RoboDK station: wcs_plc_20240624_150000.rdk

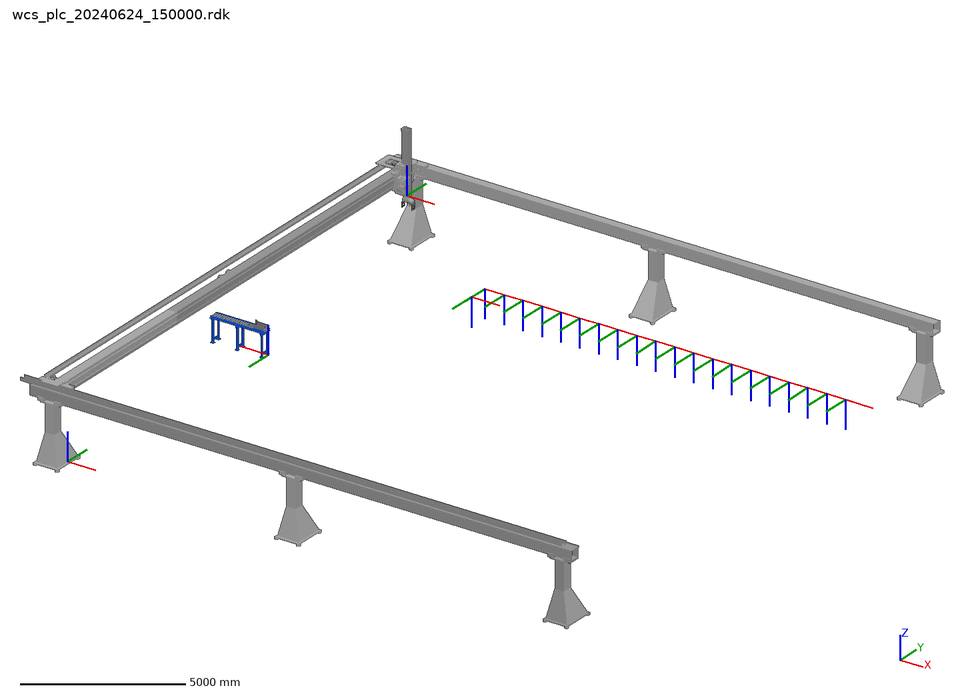
[picture v0: the station drawn from its stored meshes, robots at their saved joint values, targets as dots, program paths as lines]
Station wcs_plc_20240624_150000 (saved by RoboDK 5.6.8). Poses are relative to the parent item; angles as X-Y-Z fixed-axis rotations.
Station parameters (name, value as stored): TAGS, ['Milling']
  - frame conveyor Base at (750, 9500, 0) mm, rotated rx 0 ry 0 rz 180 deg
    - robot conveyor: 1 axes
        modified DH rows (alpha deg, a mm, theta deg, d mm): 0, 0, 0, 0 linear
        base shift (0, 0, 0) mm, rotated rx 0 ry 90 rz 0 deg
        joint limits [-99999] to [9999999]; home [0]; saved at [1000]
      - tool conveyor_TCP, TCP at (160, 110, 135) mm, rotated rx -180 ry 0 rz -180 deg
    - target con_pitch (joint target) at (1000, 0, 880) mm; joints [1000, 0, 0] of conveyor
    - target con_home (joint target) at (160, 110, 1015) mm, rotated rx -180 ry 0 rz -180 deg; joints [0] of conveyor
  - camera Camera 1
  - frame Frame 36 at (28300, 9440, 4940) mm, rotated rx -108 ry 0 rz 90 deg
  - frame gantry Base at (0, 0, 0) mm
    - robot gantry: 3 axes
        modified DH rows (alpha deg, a mm, theta deg, d mm): 0, 0, 0, 0 linear; 90, 0, 90, 0 linear; 90, 0, 0, 0 linear
        base shift (0, 0, 0) mm, rotated rx 0 ry -90 rz 180 deg
        joint limits [-5, -5, -5] to [18000, 17000, 1500]; home [0, 0, 0]; saved at [0, 0, 0]
      - frame gripper Base at (0, 0, 0) mm, rotated rx -180 ry 0 rz 0 deg
        - robot gripper: 1 axes
            modified DH rows (alpha deg, a mm, theta deg, d mm): 0, 0, 0, 0 linear
            base shift (0, 0, 0) mm, rotated rx 0 ry 90 rz 0 deg
            joint limits [-200] to [0]; home [0]; saved at [0]
        - target open_gripper (Cartesian target) at (0, 0, 0) mm; joints [0] of gripper
        - target close_gripper (Cartesian target) at (-55, 0, 0) mm; joints [-55] of gripper
      - tool gripper_TCP, TCP at (0, 0, 260) mm
    - target gantry_home (Cartesian target) at (-66.33, 17957.34, 1743.56) mm, rotated rx 180 ry 0 rz 0 deg; joints [0, 0, 0] of gantry
    - target UP_pickup (Cartesian target) at (590, 9400, 1743.56) mm, rotated rx 180 ry 0 rz 0 deg; joints [656.33, 8557.342, 0] of gantry
    - target IN_pickup (Cartesian target) at (590, 9400, 1275) mm, rotated rx 180 ry 0 rz 0 deg; joints [656.33, 8557.34, 468.56] of gantry
    - folder pallet
      - frame TeachingPoints_01-01-01 at (3833.67, 16507.34, 288.56) mm, rotated rx 180 ry 0 rz 0 deg
        - target Point_01-01-01 (Cartesian target) at (0, 0, 0) mm; joints [3900, 1450, 1195] of gantry
      - frame TeachingPoints_02-01-01 at (4533.67, 16507.34, 288.56) mm, rotated rx 180 ry 0 rz 0 deg
        - target Point_02-01-01 (Cartesian target) at (0, 0, 0) mm; joints [4600, 1450, 1195] of gantry
      - frame TeachingPoints_03-01-01 at (5233.67, 16507.34, 288.56) mm, rotated rx 180 ry 0 rz 0 deg
        - target Point_03-01-01 (Cartesian target) at (0, 0, 0) mm; joints [5300, 1450, 1195] of gantry
      - frame TeachingPoints_04-01-01 at (5933.67, 16507.34, 288.56) mm, rotated rx 180 ry 0 rz 0 deg
        - target Point_04-01-01 (Cartesian target) at (0, 0, 0) mm; joints [6000, 1450, 1195] of gantry
      - frame TeachingPoints_05-01-01 at (6633.67, 16507.34, 288.56) mm, rotated rx 180 ry 0 rz 0 deg
        - target Point_05-01-01 (Cartesian target) at (0, 0, 0) mm; joints [6700, 1450, 1195] of gantry
      - frame TeachingPoints_06-01-01 at (7333.67, 16507.34, 288.56) mm, rotated rx 180 ry 0 rz 0 deg
        - target Point_06-01-01 (Cartesian target) at (0, 0, 0) mm; joints [7400, 1450, 1195] of gantry
      - frame TeachingPoints_07-01-01 at (8033.67, 16507.34, 288.56) mm, rotated rx 180 ry 0 rz 0 deg
        - target Point_07-01-01 (Cartesian target) at (0, 0, 0) mm; joints [8100, 1450, 1195] of gantry
      - frame TeachingPoints_08-01-01 at (8733.67, 16507.34, 288.56) mm, rotated rx 180 ry 0 rz 0 deg
        - target Point_08-01-01 (Cartesian target) at (0, 0, 0) mm; joints [8800, 1450, 1195] of gantry
      - frame TeachingPoints_09-01-01 at (9433.67, 16507.34, 288.56) mm, rotated rx 180 ry 0 rz 0 deg
        - target Point_09-01-01 (Cartesian target) at (0, 0, 0) mm; joints [9500, 1450, 1195] of gantry
      - frame TeachingPoints_10-01-01 at (10133.67, 16507.34, 288.56) mm, rotated rx 180 ry 0 rz 0 deg
        - target Point_10-01-01 (Cartesian target) at (0, 0, 0) mm; joints [10200, 1450, 1195] of gantry
      - frame TeachingPoints_11-01-01 at (10833.67, 16507.34, 288.56) mm, rotated rx 180 ry 0 rz 0 deg
        - target Point_11-01-01 (Cartesian target) at (0, 0, 0) mm; joints [10900, 1450, 1195] of gantry
      - frame TeachingPoints_12-01-01 at (11533.67, 16507.34, 288.56) mm, rotated rx 180 ry 0 rz 0 deg
        - target Point_12-01-01 (Cartesian target) at (0, 0, 0) mm; joints [11600, 1450, 1195] of gantry
      - frame TeachingPoints_13-01-01 at (12233.67, 16507.34, 288.56) mm, rotated rx 180 ry 0 rz 0 deg
        - target Point_13-01-01 (Cartesian target) at (0, 0, 0) mm; joints [12300, 1450, 1195] of gantry
      - frame TeachingPoints_14-01-01 at (12933.67, 16507.34, 288.56) mm, rotated rx 180 ry 0 rz 0 deg
        - target Point_14-01-01 (Cartesian target) at (0, 0, 0) mm; joints [13000, 1450, 1195] of gantry
      - frame TeachingPoints_15-01-01 at (13633.67, 16507.34, 288.56) mm, rotated rx 180 ry 0 rz 0 deg
        - target Point_15-01-01 (Cartesian target) at (0, 0, 0) mm; joints [13700, 1450, 1195] of gantry
      - frame TeachingPoints_16-01-01 at (14333.67, 16507.34, 288.56) mm, rotated rx 180 ry 0 rz 0 deg
        - target Point_16-01-01 (Cartesian target) at (0, 0, 0) mm; joints [14400, 1450, 1195] of gantry
      - frame TeachingPoints_17-01-01 at (15033.67, 16507.34, 288.56) mm, rotated rx 180 ry 0 rz 0 deg
        - target Point_17-01-01 (Cartesian target) at (0, 0, 0) mm; joints [15100, 1450, 1195] of gantry
      - frame TeachingPoints_18-01-01 at (15733.67, 16507.34, 288.56) mm, rotated rx 180 ry 0 rz 0 deg
        - target Point_18-01-01 (Cartesian target) at (0, 0, 0) mm; joints [15800, 1450, 1195] of gantry
      - frame TeachingPoints_19-01-01 at (16433.67, 16507.34, 288.56) mm, rotated rx 180 ry 0 rz 0 deg
        - target Point_19-01-01 (Cartesian target) at (0, 0, 0) mm; joints [16500, 1450, 1195] of gantry
      - frame TeachingPoints_20-01-01 at (17133.67, 16507.34, 288.56) mm, rotated rx 180 ry 0 rz 0 deg
        - target Point_20-01-01 (Cartesian target) at (0, 0, 0) mm; joints [17200, 1450, 1195] of gantry
      - frame TeachingPoints_01-02-01 at (3833.67, 15807.34, 288.56) mm, rotated rx 180 ry 0 rz 0 deg
        - target Point_01-02-01 (Cartesian target) at (0, 0, 0) mm; joints [3900, 2150, 1195] of gantry
      - frame TeachingPoints_02-02-01 at (4533.67, 15807.34, 288.56) mm, rotated rx 180 ry 0 rz 0 deg
        - target Point_02-02-01 (Cartesian target) at (0, 0, 0) mm; joints [4600, 2150, 1195] of gantry
      - frame TeachingPoints_03-02-01 at (5233.67, 15807.34, 288.56) mm, rotated rx 180 ry 0 rz 0 deg
        - target Point_03-02-01 (Cartesian target) at (0, 0, 0) mm; joints [5300, 2150, 1195] of gantry
      - frame TeachingPoints_04-02-01 at (5933.67, 15807.34, 288.56) mm, rotated rx 180 ry 0 rz 0 deg
        - target Point_04-02-01 (Cartesian target) at (0, 0, 0) mm; joints [6000, 2150, 1195] of gantry
      - frame TeachingPoints_05-02-01 at (6633.67, 15807.34, 288.56) mm, rotated rx 180 ry 0 rz 0 deg
        - target Point_05-02-01 (Cartesian target) at (0, 0, 0) mm; joints [6700, 2150, 1195] of gantry
      - frame TeachingPoints_06-02-01 at (7333.67, 15807.34, 288.56) mm, rotated rx 180 ry 0 rz 0 deg
        - target Point_06-02-01 (Cartesian target) at (0, 0, 0) mm; joints [7400, 2150, 1195] of gantry
      - frame TeachingPoints_07-02-01 at (8033.67, 15807.34, 288.56) mm, rotated rx 180 ry 0 rz 0 deg
        - target Point_07-02-01 (Cartesian target) at (0, 0, 0) mm; joints [8100, 2150, 1195] of gantry
      - frame TeachingPoints_08-02-01 at (8733.67, 15807.34, 288.56) mm, rotated rx 180 ry 0 rz 0 deg
        - target Point_08-02-01 (Cartesian target) at (0, 0, 0) mm; joints [8800, 2150, 1195] of gantry
      - frame TeachingPoints_09-02-01 at (9433.67, 15807.34, 288.56) mm, rotated rx 180 ry 0 rz 0 deg
        - target Point_09-02-01 (Cartesian target) at (0, 0, 0) mm; joints [9500, 2150, 1195] of gantry
      - frame TeachingPoints_10-02-01 at (10133.67, 15807.34, 288.56) mm, rotated rx 180 ry 0 rz 0 deg
        - target Point_10-02-01 (Cartesian target) at (0, 0, 0) mm; joints [10200, 2150, 1195] of gantry
      - frame TeachingPoints_11-02-01 at (10833.67, 15807.34, 288.56) mm, rotated rx 180 ry 0 rz 0 deg
        - target Point_11-02-01 (Cartesian target) at (0, 0, 0) mm; joints [10900, 2150, 1195] of gantry
      - frame TeachingPoints_12-02-01 at (11533.67, 15807.34, 288.56) mm, rotated rx 180 ry 0 rz 0 deg
        - target Point_12-02-01 (Cartesian target) at (0, 0, 0) mm; joints [11600, 2150, 1195] of gantry
      - frame TeachingPoints_13-02-01 at (12233.67, 15807.34, 288.56) mm, rotated rx 180 ry 0 rz 0 deg
        - target Point_13-02-01 (Cartesian target) at (0, 0, 0) mm; joints [12300, 2150, 1195] of gantry
      - frame TeachingPoints_14-02-01 at (12933.67, 15807.34, 288.56) mm, rotated rx 180 ry 0 rz 0 deg
        - target Point_14-02-01 (Cartesian target) at (0, 0, 0) mm; joints [13000, 2150, 1195] of gantry
      - frame TeachingPoints_15-02-01 at (13633.67, 15807.34, 288.56) mm, rotated rx 180 ry 0 rz 0 deg
        - target Point_15-02-01 (Cartesian target) at (0, 0, 0) mm; joints [13700, 2150, 1195] of gantry
      - frame TeachingPoints_16-02-01 at (14333.67, 15807.34, 288.56) mm, rotated rx 180 ry 0 rz 0 deg
        - target Point_16-02-01 (Cartesian target) at (0, 0, 0) mm; joints [14400, 2150, 1195] of gantry
      - frame TeachingPoints_17-02-01 at (15033.67, 15807.34, 288.56) mm, rotated rx 180 ry 0 rz 0 deg
        - target Point_17-02-01 (Cartesian target) at (0, 0, 0) mm; joints [15100, 2150, 1195] of gantry
      - frame TeachingPoints_18-02-01 at (15733.67, 15807.34, 288.56) mm, rotated rx 180 ry 0 rz 0 deg
        - target Point_18-02-01 (Cartesian target) at (0, 0, 0) mm; joints [15800, 2150, 1195] of gantry
      - frame TeachingPoints_19-02-01 at (16433.67, 15807.34, 288.56) mm, rotated rx 180 ry 0 rz 0 deg
        - target Point_19-02-01 (Cartesian target) at (0, 0, 0) mm; joints [16500, 2150, 1195] of gantry
      - frame TeachingPoints_20-02-01 at (17133.67, 15807.34, 288.56) mm, rotated rx 180 ry 0 rz 0 deg
        - target Point_20-02-01 (Cartesian target) at (0, 0, 0) mm; joints [17200, 2150, 1195] of gantry
      - frame TeachingPoints_01-03-01 at (3833.67, 15107.34, 288.56) mm, rotated rx 180 ry 0 rz 0 deg
        - target Point_01-03-01 (Cartesian target) at (0, 0, 0) mm; joints [3900, 2850, 1195] of gantry
      - frame TeachingPoints_02-03-01 at (4533.67, 15107.34, 288.56) mm, rotated rx 180 ry 0 rz 0 deg
        - target Point_02-03-01 (Cartesian target) at (0, 0, 0) mm; joints [4600, 2850, 1195] of gantry
      - frame TeachingPoints_03-03-01 at (5233.67, 15107.34, 288.56) mm, rotated rx 180 ry 0 rz 0 deg
        - target Point_03-03-01 (Cartesian target) at (0, 0, 0) mm; joints [5300, 2850, 1195] of gantry
      - frame TeachingPoints_04-03-01 at (5933.67, 15107.34, 288.56) mm, rotated rx 180 ry 0 rz 0 deg
        - target Point_04-03-01 (Cartesian target) at (0, 0, 0) mm; joints [6000, 2850, 1195] of gantry
      - frame TeachingPoints_05-03-01 at (6633.67, 15107.34, 288.56) mm, rotated rx 180 ry 0 rz 0 deg
        - target Point_05-03-01 (Cartesian target) at (0, 0, 0) mm; joints [6700, 2850, 1195] of gantry
      - frame TeachingPoints_06-03-01 at (7333.67, 15107.34, 288.56) mm, rotated rx 180 ry 0 rz 0 deg
        - target Point_06-03-01 (Cartesian target) at (0, 0, 0) mm; joints [7400, 2850, 1195] of gantry
      - frame TeachingPoints_07-03-01 at (8033.67, 15107.34, 288.56) mm, rotated rx 180 ry 0 rz 0 deg
        - target Point_07-03-01 (Cartesian target) at (0, 0, 0) mm; joints [8100, 2850, 1195] of gantry
      - frame TeachingPoints_08-03-01 at (8733.67, 15107.34, 288.56) mm, rotated rx 180 ry 0 rz 0 deg
        - target Point_08-03-01 (Cartesian target) at (0, 0, 0) mm; joints [8800, 2850, 1195] of gantry
      - frame TeachingPoints_09-03-01 at (9433.67, 15107.34, 288.56) mm, rotated rx 180 ry 0 rz 0 deg
        - target Point_09-03-01 (Cartesian target) at (0, 0, 0) mm; joints [9500, 2850, 1195] of gantry
      - frame TeachingPoints_10-03-01 at (10133.67, 15107.34, 288.56) mm, rotated rx 180 ry 0 rz 0 deg
        - target Point_10-03-01 (Cartesian target) at (0, 0, 0) mm; joints [10200, 2850, 1195] of gantry
      - frame TeachingPoints_11-03-01 at (10833.67, 15107.34, 288.56) mm, rotated rx 180 ry 0 rz 0 deg
        - target Point_11-03-01 (Cartesian target) at (0, 0, 0) mm; joints [10900, 2850, 1195] of gantry
      - frame TeachingPoints_12-03-01 at (11533.67, 15107.34, 288.56) mm, rotated rx 180 ry 0 rz 0 deg
        - target Point_12-03-01 (Cartesian target) at (0, 0, 0) mm; joints [11600, 2850, 1195] of gantry
      - frame TeachingPoints_13-03-01 at (12233.67, 15107.34, 288.56) mm, rotated rx 180 ry 0 rz 0 deg
        - target Point_13-03-01 (Cartesian target) at (0, 0, 0) mm; joints [12300, 2850, 1195] of gantry
      - frame TeachingPoints_14-03-01 at (12933.67, 15107.34, 288.56) mm, rotated rx 180 ry 0 rz 0 deg
        - target Point_14-03-01 (Cartesian target) at (0, 0, 0) mm; joints [13000, 2850, 1195] of gantry
      - frame TeachingPoints_15-03-01 at (13633.67, 15107.34, 288.56) mm, rotated rx 180 ry 0 rz 0 deg
        - target Point_15-03-01 (Cartesian target) at (0, 0, 0) mm; joints [13700, 2850, 1195] of gantry
      - frame TeachingPoints_16-03-01 at (14333.67, 15107.34, 288.56) mm, rotated rx 180 ry 0 rz 0 deg
        - target Point_16-03-01 (Cartesian target) at (0, 0, 0) mm; joints [14400, 2850, 1195] of gantry
      - frame TeachingPoints_17-03-01 at (15033.67, 15107.34, 288.56) mm, rotated rx 180 ry 0 rz 0 deg
        - target Point_17-03-01 (Cartesian target) at (0, 0, 0) mm; joints [15100, 2850, 1195] of gantry
      - frame TeachingPoints_18-03-01 at (15733.67, 15107.34, 288.56) mm, rotated rx 180 ry 0 rz 0 deg
        - target Point_18-03-01 (Cartesian target) at (0, 0, 0) mm; joints [15800, 2850, 1195] of gantry
      - frame TeachingPoints_19-03-01 at (16433.67, 15107.34, 288.56) mm, rotated rx 180 ry 0 rz 0 deg
        - target Point_19-03-01 (Cartesian target) at (0, 0, 0) mm; joints [16500, 2850, 1195] of gantry
      - frame TeachingPoints_20-03-01 at (17133.67, 15107.34, 288.56) mm, rotated rx 180 ry 0 rz 0 deg
        - target Point_20-03-01 (Cartesian target) at (0, 0, 0) mm; joints [17200, 2850, 1195] of gantry
      - frame TeachingPoints_01-04-01 at (3833.67, 14407.34, 288.56) mm, rotated rx 180 ry 0 rz 0 deg
        - target Point_01-04-01 (Cartesian target) at (0, 0, 0) mm; joints [3900, 3550, 1195] of gantry
      - frame TeachingPoints_02-04-01 at (4533.67, 14407.34, 288.56) mm, rotated rx 180 ry 0 rz 0 deg
        - target Point_02-04-01 (Cartesian target) at (0, 0, 0) mm; joints [4600, 3550, 1195] of gantry
      - frame TeachingPoints_03-04-01 at (5233.67, 14407.34, 288.56) mm, rotated rx 180 ry 0 rz 0 deg
        - target Point_03-04-01 (Cartesian target) at (0, 0, 0) mm; joints [5300, 3550, 1195] of gantry
      - frame TeachingPoints_04-04-01 at (5933.67, 14407.34, 288.56) mm, rotated rx 180 ry 0 rz 0 deg
        - target Point_04-04-01 (Cartesian target) at (0, 0, 0) mm; joints [6000, 3550, 1195] of gantry
      - frame TeachingPoints_05-04-01 at (6633.67, 14407.34, 288.56) mm, rotated rx 180 ry 0 rz 0 deg
        - target Point_05-04-01 (Cartesian target) at (0, 0, 0) mm; joints [6700, 3550, 1195] of gantry
      - frame TeachingPoints_06-04-01 at (7333.67, 14407.34, 288.56) mm, rotated rx 180 ry 0 rz 0 deg
        - target Point_06-04-01 (Cartesian target) at (0, 0, 0) mm; joints [7400, 3550, 1195] of gantry
      - frame TeachingPoints_07-04-01 at (8033.67, 14407.34, 288.56) mm, rotated rx 180 ry 0 rz 0 deg
        - target Point_07-04-01 (Cartesian target) at (0, 0, 0) mm; joints [8100, 3550, 1195] of gantry
      - frame TeachingPoints_08-04-01 at (8733.67, 14407.34, 288.56) mm, rotated rx 180 ry 0 rz 0 deg
        - target Point_08-04-01 (Cartesian target) at (0, 0, 0) mm; joints [8800, 3550, 1195] of gantry
      - frame TeachingPoints_09-04-01 at (9433.67, 14407.34, 288.56) mm, rotated rx 180 ry 0 rz 0 deg
        - target Point_09-04-01 (Cartesian target) at (0, 0, 0) mm; joints [9500, 3550, 1195] of gantry
      - frame TeachingPoints_10-04-01 at (10133.67, 14407.34, 288.56) mm, rotated rx 180 ry 0 rz 0 deg
        - target Point_10-04-01 (Cartesian target) at (0, 0, 0) mm; joints [10200, 3550, 1195] of gantry
      - frame TeachingPoints_11-04-01 at (10833.67, 14407.34, 288.56) mm, rotated rx 180 ry 0 rz 0 deg
        - target Point_11-04-01 (Cartesian target) at (0, 0, 0) mm; joints [10900, 3550, 1195] of gantry
      - frame TeachingPoints_12-04-01 at (11533.67, 14407.34, 288.56) mm, rotated rx 180 ry 0 rz 0 deg
        - target Point_12-04-01 (Cartesian target) at (0, 0, 0) mm; joints [11600, 3550, 1195] of gantry
      - frame TeachingPoints_13-04-01 at (12233.67, 14407.34, 288.56) mm, rotated rx 180 ry 0 rz 0 deg
        - target Point_13-04-01 (Cartesian target) at (0, 0, 0) mm; joints [12300, 3550, 1195] of gantry
      - frame TeachingPoints_14-04-01 at (12933.67, 14407.34, 288.56) mm, rotated rx 180 ry 0 rz 0 deg
        - target Point_14-04-01 (Cartesian target) at (0, 0, 0) mm; joints [13000, 3550, 1195] of gantry
      - frame TeachingPoints_15-04-01 at (13633.67, 14407.34, 288.56) mm, rotated rx 180 ry 0 rz 0 deg
        - target Point_15-04-01 (Cartesian target) at (0, 0, 0) mm; joints [13700, 3550, 1195] of gantry
      - frame TeachingPoints_16-04-01 at (14333.67, 14407.34, 288.56) mm, rotated rx 180 ry 0 rz 0 deg
        - target Point_16-04-01 (Cartesian target) at (0, 0, 0) mm; joints [14400, 3550, 1195] of gantry
      - frame TeachingPoints_17-04-01 at (15033.67, 14407.34, 288.56) mm, rotated rx 180 ry 0 rz 0 deg
        - target Point_17-04-01 (Cartesian target) at (0, 0, 0) mm; joints [15100, 3550, 1195] of gantry
      - frame TeachingPoints_18-04-01 at (15733.67, 14407.34, 288.56) mm, rotated rx 180 ry 0 rz 0 deg
        - target Point_18-04-01 (Cartesian target) at (0, 0, 0) mm; joints [15800, 3550, 1195] of gantry
      - frame TeachingPoints_19-04-01 at (16433.67, 14407.34, 288.56) mm, rotated rx 180 ry 0 rz 0 deg
        - target Point_19-04-01 (Cartesian target) at (0, 0, 0) mm; joints [16500, 3550, 1195] of gantry
      - frame TeachingPoints_20-04-01 at (17133.67, 14407.34, 288.56) mm, rotated rx 180 ry 0 rz 0 deg
        - target Point_20-04-01 (Cartesian target) at (0, 0, 0) mm; joints [17200, 3550, 1195] of gantry
      - frame TeachingPoints_01-05-01 at (3833.67, 13707.34, 288.56) mm, rotated rx 180 ry 0 rz 0 deg
        - target Point_01-05-01 (Cartesian target) at (0, 0, 0) mm; joints [3900, 4250, 1195] of gantry
      - frame TeachingPoints_02-05-01 at (4533.67, 13707.34, 288.56) mm, rotated rx 180 ry 0 rz 0 deg
        - target Point_02-05-01 (Cartesian target) at (0, 0, 0) mm; joints [4600, 4250, 1195] of gantry
      - frame TeachingPoints_03-05-01 at (5233.67, 13707.34, 288.56) mm, rotated rx 180 ry 0 rz 0 deg
        - target Point_03-05-01 (Cartesian target) at (0, 0, 0) mm; joints [5300, 4250, 1195] of gantry
      - frame TeachingPoints_04-05-01 at (5933.67, 13707.34, 288.56) mm, rotated rx 180 ry 0 rz 0 deg
        - target Point_04-05-01 (Cartesian target) at (0, 0, 0) mm; joints [6000, 4250, 1195] of gantry
      - frame TeachingPoints_05-05-01 at (6633.67, 13707.34, 288.56) mm, rotated rx 180 ry 0 rz 0 deg
        - target Point_05-05-01 (Cartesian target) at (0, 0, 0) mm; joints [6700, 4250, 1195] of gantry
      - frame TeachingPoints_06-05-01 at (7333.67, 13707.34, 288.56) mm, rotated rx 180 ry 0 rz 0 deg
        - target Point_06-05-01 (Cartesian target) at (0, 0, 0) mm; joints [7400, 4250, 1195] of gantry
      - frame TeachingPoints_07-05-01 at (8033.67, 13707.34, 288.56) mm, rotated rx 180 ry 0 rz 0 deg
        - target Point_07-05-01 (Cartesian target) at (0, 0, 0) mm; joints [8100, 4250, 1195] of gantry
      - frame TeachingPoints_08-05-01 at (8733.67, 13707.34, 288.56) mm, rotated rx 180 ry 0 rz 0 deg
        - target Point_08-05-01 (Cartesian target) at (0, 0, 0) mm; joints [8800, 4250, 1195] of gantry
      - frame TeachingPoints_09-05-01 at (9433.67, 13707.34, 288.56) mm, rotated rx 180 ry 0 rz 0 deg
        - target Point_09-05-01 (Cartesian target) at (0, 0, 0) mm; joints [9500, 4250, 1195] of gantry
      - frame TeachingPoints_10-05-01 at (10133.67, 13707.34, 288.56) mm, rotated rx 180 ry 0 rz 0 deg
        - target Point_10-05-01 (Cartesian target) at (0, 0, 0) mm; joints [10200, 4250, 1195] of gantry
      - frame TeachingPoints_11-05-01 at (10833.67, 13707.34, 288.56) mm, rotated rx 180 ry 0 rz 0 deg
        - target Point_11-05-01 (Cartesian target) at (0, 0, 0) mm; joints [10900, 4250, 1195] of gantry
      - frame TeachingPoints_12-05-01 at (11533.67, 13707.34, 288.56) mm, rotated rx 180 ry 0 rz 0 deg
        - target Point_12-05-01 (Cartesian target) at (0, 0, 0) mm; joints [11600, 4250, 1195] of gantry
      - frame TeachingPoints_13-05-01 at (12233.67, 13707.34, 288.56) mm, rotated rx 180 ry 0 rz 0 deg
        - target Point_13-05-01 (Cartesian target) at (0, 0, 0) mm; joints [12300, 4250, 1195] of gantry
      - frame TeachingPoints_14-05-01 at (12933.67, 13707.34, 288.56) mm, rotated rx 180 ry 0 rz 0 deg
        - target Point_14-05-01 (Cartesian target) at (0, 0, 0) mm; joints [13000, 4250, 1195] of gantry
      - frame TeachingPoints_15-05-01 at (13633.67, 13707.34, 288.56) mm, rotated rx 180 ry 0 rz 0 deg
        - target Point_15-05-01 (Cartesian target) at (0, 0, 0) mm; joints [13700, 4250, 1195] of gantry
      - frame TeachingPoints_16-05-01 at (14333.67, 13707.34, 288.56) mm, rotated rx 180 ry 0 rz 0 deg
        - target Point_16-05-01 (Cartesian target) at (0, 0, 0) mm; joints [14400, 4250, 1195] of gantry
      - frame TeachingPoints_17-05-01 at (15033.67, 13707.34, 288.56) mm, rotated rx 180 ry 0 rz 0 deg
        - target Point_17-05-01 (Cartesian target) at (0, 0, 0) mm; joints [15100, 4250, 1195] of gantry
      - frame TeachingPoints_18-05-01 at (15733.67, 13707.34, 288.56) mm, rotated rx 180 ry 0 rz 0 deg
        - target Point_18-05-01 (Cartesian target) at (0, 0, 0) mm; joints [15800, 4250, 1195] of gantry
      - frame TeachingPoints_19-05-01 at (16433.67, 13707.34, 288.56) mm, rotated rx 180 ry 0 rz 0 deg
        - target Point_19-05-01 (Cartesian target) at (0, 0, 0) mm; joints [16500, 4250, 1195] of gantry
      - frame TeachingPoints_20-05-01 at (17133.67, 13707.34, 288.56) mm, rotated rx 180 ry 0 rz 0 deg
        - target Point_20-05-01 (Cartesian target) at (0, 0, 0) mm; joints [17200, 4250, 1195] of gantry
      - frame TeachingPoints_01-06-01 at (3833.67, 13007.34, 288.56) mm, rotated rx 180 ry 0 rz 0 deg
        - target Point_01-06-01 (Cartesian target) at (0, 0, 0) mm; joints [3900, 4950, 1195] of gantry
      - frame TeachingPoints_02-06-01 at (4533.67, 13007.34, 288.56) mm, rotated rx 180 ry 0 rz 0 deg
        - target Point_02-06-01 (Cartesian target) at (0, 0, 0) mm; joints [4600, 4950, 1195] of gantry
      - frame TeachingPoints_03-06-01 at (5233.67, 13007.34, 288.56) mm, rotated rx 180 ry 0 rz 0 deg
        - target Point_03-06-01 (Cartesian target) at (0, 0, 0) mm; joints [5300, 4950, 1195] of gantry
      - frame TeachingPoints_04-06-01 at (5933.67, 13007.34, 288.56) mm, rotated rx 180 ry 0 rz 0 deg
        - target Point_04-06-01 (Cartesian target) at (0, 0, 0) mm; joints [6000, 4950, 1195] of gantry
      - frame TeachingPoints_05-06-01 at (6633.67, 13007.34, 288.56) mm, rotated rx 180 ry 0 rz 0 deg
        - target Point_05-06-01 (Cartesian target) at (0, 0, 0) mm; joints [6700, 4950, 1195] of gantry
      - frame TeachingPoints_06-06-01 at (7333.67, 13007.34, 288.56) mm, rotated rx 180 ry 0 rz 0 deg
        - target Point_06-06-01 (Cartesian target) at (0, 0, 0) mm; joints [7400, 4950, 1195] of gantry
      - frame TeachingPoints_07-06-01 at (8033.67, 13007.34, 288.56) mm, rotated rx 180 ry 0 rz 0 deg
        - target Point_07-06-01 (Cartesian target) at (0, 0, 0) mm; joints [8100, 4950, 1195] of gantry
      - frame TeachingPoints_08-06-01 at (8733.67, 13007.34, 288.56) mm, rotated rx 180 ry 0 rz 0 deg
        - target Point_08-06-01 (Cartesian target) at (0, 0, 0) mm; joints [8800, 4950, 1195] of gantry
      - frame TeachingPoints_09-06-01 at (9433.67, 13007.34, 288.56) mm, rotated rx 180 ry 0 rz 0 deg
        - target Point_09-06-01 (Cartesian target) at (0, 0, 0) mm; joints [9500, 4950, 1195] of gantry
      - frame TeachingPoints_10-06-01 at (10133.67, 13007.34, 288.56) mm, rotated rx 180 ry 0 rz 0 deg
        - target Point_10-06-01 (Cartesian target) at (0, 0, 0) mm; joints [10200, 4950, 1195] of gantry
      - frame TeachingPoints_11-06-01 at (10833.67, 13007.34, 288.56) mm, rotated rx 180 ry 0 rz 0 deg
        - target Point_11-06-01 (Cartesian target) at (0, 0, 0) mm; joints [10900, 4950, 1195] of gantry
      - frame TeachingPoints_12-06-01 at (11533.67, 13007.34, 288.56) mm, rotated rx 180 ry 0 rz 0 deg
        - target Point_12-06-01 (Cartesian target) at (0, 0, 0) mm; joints [11600, 4950, 1195] of gantry
      - frame TeachingPoints_13-06-01 at (12233.67, 13007.34, 288.56) mm, rotated rx 180 ry 0 rz 0 deg
        - target Point_13-06-01 (Cartesian target) at (0, 0, 0) mm; joints [12300, 4950, 1195] of gantry
      - frame TeachingPoints_14-06-01 at (12933.67, 13007.34, 288.56) mm, rotated rx 180 ry 0 rz 0 deg
        - target Point_14-06-01 (Cartesian target) at (0, 0, 0) mm; joints [13000, 4950, 1195] of gantry
      - frame TeachingPoints_15-06-01 at (13633.67, 13007.34, 288.56) mm, rotated rx 180 ry 0 rz 0 deg
        - target Point_15-06-01 (Cartesian target) at (0, 0, 0) mm; joints [13700, 4950, 1195] of gantry
      - frame TeachingPoints_16-06-01 at (14333.67, 13007.34, 288.56) mm, rotated rx 180 ry 0 rz 0 deg
        - target Point_16-06-01 (Cartesian target) at (0, 0, 0) mm; joints [14400, 4950, 1195] of gantry
      - frame TeachingPoints_17-06-01 at (15033.67, 13007.34, 288.56) mm, rotated rx 180 ry 0 rz 0 deg
        - target Point_17-06-01 (Cartesian target) at (0, 0, 0) mm; joints [15100, 4950, 1195] of gantry
      - frame TeachingPoints_18-06-01 at (15733.67, 13007.34, 288.56) mm, rotated rx 180 ry 0 rz 0 deg
        - target Point_18-06-01 (Cartesian target) at (0, 0, 0) mm; joints [15800, 4950, 1195] of gantry
      - frame TeachingPoints_19-06-01 at (16433.67, 13007.34, 288.56) mm, rotated rx 180 ry 0 rz 0 deg
        - target Point_19-06-01 (Cartesian target) at (0, 0, 0) mm; joints [16500, 4950, 1195] of gantry
      - frame TeachingPoints_20-06-01 at (17133.67, 13007.34, 288.56) mm, rotated rx 180 ry 0 rz 0 deg
        - target Point_20-06-01 (Cartesian target) at (0, 0, 0) mm; joints [17200, 4950, 1195] of gantry
      - frame TeachingPoints_01-07-01 at (3833.67, 12307.34, 288.56) mm, rotated rx 180 ry 0 rz 0 deg
        - target Point_01-07-01 (Cartesian target) at (0, 0, 0) mm; joints [3900, 5650, 1195] of gantry
      - frame TeachingPoints_02-07-01 at (4533.67, 12307.34, 288.56) mm, rotated rx 180 ry 0 rz 0 deg
        - target Point_02-07-01 (Cartesian target) at (0, 0, 0) mm; joints [4600, 5650, 1195] of gantry
      - frame TeachingPoints_03-07-01 at (5233.67, 12307.34, 288.56) mm, rotated rx 180 ry 0 rz 0 deg
        - target Point_03-07-01 (Cartesian target) at (0, 0, 0) mm; joints [5300, 5650, 1195] of gantry
      - frame TeachingPoints_04-07-01 at (5933.67, 12307.34, 288.56) mm, rotated rx 180 ry 0 rz 0 deg
        - target Point_04-07-01 (Cartesian target) at (0, 0, 0) mm; joints [6000, 5650, 1195] of gantry
      - frame TeachingPoints_05-07-01 at (6633.67, 12307.34, 288.56) mm, rotated rx 180 ry 0 rz 0 deg
        - target Point_05-07-01 (Cartesian target) at (0, 0, 0) mm; joints [6700, 5650, 1195] of gantry
      - frame TeachingPoints_06-07-01 at (7333.67, 12307.34, 288.56) mm, rotated rx 180 ry 0 rz 0 deg
        - target Point_06-07-01 (Cartesian target) at (0, 0, 0) mm; joints [7400, 5650, 1195] of gantry
      - frame TeachingPoints_07-07-01 at (8033.67, 12307.34, 288.56) mm, rotated rx 180 ry 0 rz 0 deg
        - target Point_07-07-01 (Cartesian target) at (0, 0, 0) mm; joints [8100, 5650, 1195] of gantry
      - frame TeachingPoints_08-07-01 at (8733.67, 12307.34, 288.56) mm, rotated rx 180 ry 0 rz 0 deg
        - target Point_08-07-01 (Cartesian target) at (0, 0, 0) mm; joints [8800, 5650, 1195] of gantry
      - frame TeachingPoints_09-07-01 at (9433.67, 12307.34, 288.56) mm, rotated rx 180 ry 0 rz 0 deg
        - target Point_09-07-01 (Cartesian target) at (0, 0, 0) mm; joints [9500, 5650, 1195] of gantry
      - frame TeachingPoints_10-07-01 at (10133.67, 12307.34, 288.56) mm, rotated rx 180 ry 0 rz 0 deg
        - target Point_10-07-01 (Cartesian target) at (0, 0, 0) mm; joints [10200, 5650, 1195] of gantry
      - frame TeachingPoints_11-07-01 at (10833.67, 12307.34, 288.56) mm, rotated rx 180 ry 0 rz 0 deg
        - target Point_11-07-01 (Cartesian target) at (0, 0, 0) mm; joints [10900, 5650, 1195] of gantry
      - frame TeachingPoints_12-07-01 at (11533.67, 12307.34, 288.56) mm, rotated rx 180 ry 0 rz 0 deg
        - target Point_12-07-01 (Cartesian target) at (0, 0, 0) mm; joints [11600, 5650, 1195] of gantry
      - frame TeachingPoints_13-07-01 at (12233.67, 12307.34, 288.56) mm, rotated rx 180 ry 0 rz 0 deg
        - target Point_13-07-01 (Cartesian target) at (0, 0, 0) mm; joints [12300, 5650, 1195] of gantry
      - frame TeachingPoints_14-07-01 at (12933.67, 12307.34, 288.56) mm, rotated rx 180 ry 0 rz 0 deg
        - target Point_14-07-01 (Cartesian target) at (0, 0, 0) mm; joints [13000, 5650, 1195] of gantry
      - frame TeachingPoints_15-07-01 at (13633.67, 12307.34, 288.56) mm, rotated rx 180 ry 0 rz 0 deg
        - target Point_15-07-01 (Cartesian target) at (0, 0, 0) mm; joints [13700, 5650, 1195] of gantry
      - frame TeachingPoints_16-07-01 at (14333.67, 12307.34, 288.56) mm, rotated rx 180 ry 0 rz 0 deg
        - target Point_16-07-01 (Cartesian target) at (0, 0, 0) mm; joints [14400, 5650, 1195] of gantry
      - frame TeachingPoints_17-07-01 at (15033.67, 12307.34, 288.56) mm, rotated rx 180 ry 0 rz 0 deg
        - target Point_17-07-01 (Cartesian target) at (0, 0, 0) mm; joints [15100, 5650, 1195] of gantry
      - frame TeachingPoints_18-07-01 at (15733.67, 12307.34, 288.56) mm, rotated rx 180 ry 0 rz 0 deg
        - target Point_18-07-01 (Cartesian target) at (0, 0, 0) mm; joints [15800, 5650, 1195] of gantry
      - frame TeachingPoints_19-07-01 at (16433.67, 12307.34, 288.56) mm, rotated rx 180 ry 0 rz 0 deg
        - target Point_19-07-01 (Cartesian target) at (0, 0, 0) mm; joints [16500, 5650, 1195] of gantry
      - frame TeachingPoints_20-07-01 at (17133.67, 12307.34, 288.56) mm, rotated rx 180 ry 0 rz 0 deg
        - target Point_20-07-01 (Cartesian target) at (0, 0, 0) mm; joints [17200, 5650, 1195] of gantry
      - frame TeachingPoints_01-08-01 at (3833.67, 11607.34, 288.56) mm, rotated rx 180 ry 0 rz 0 deg
        - target Point_01-08-01 (Cartesian target) at (0, 0, 0) mm; joints [3900, 6350, 1195] of gantry
      - frame TeachingPoints_02-08-01 at (4533.67, 11607.34, 288.56) mm, rotated rx 180 ry 0 rz 0 deg
        - target Point_02-08-01 (Cartesian target) at (0, 0, 0) mm; joints [4600, 6350, 1195] of gantry
      - frame TeachingPoints_03-08-01 at (5233.67, 11607.34, 288.56) mm, rotated rx 180 ry 0 rz 0 deg
        - target Point_03-08-01 (Cartesian target) at (0, 0, 0) mm; joints [5300, 6350, 1195] of gantry
      - frame TeachingPoints_04-08-01 at (5933.67, 11607.34, 288.56) mm, rotated rx 180 ry 0 rz 0 deg
        - target Point_04-08-01 (Cartesian target) at (0, 0, 0) mm; joints [6000, 6350, 1195] of gantry
      - frame TeachingPoints_05-08-01 at (6633.67, 11607.34, 288.56) mm, rotated rx 180 ry 0 rz 0 deg
        - target Point_05-08-01 (Cartesian target) at (0, 0, 0) mm; joints [6700, 6350, 1195] of gantry
      - frame TeachingPoints_06-08-01 at (7333.67, 11607.34, 288.56) mm, rotated rx 180 ry 0 rz 0 deg
        - target Point_06-08-01 (Cartesian target) at (0, 0, 0) mm; joints [7400, 6350, 1195] of gantry
      - frame TeachingPoints_07-08-01 at (8033.67, 11607.34, 288.56) mm, rotated rx 180 ry 0 rz 0 deg
        - target Point_07-08-01 (Cartesian target) at (0, 0, 0) mm; joints [8100, 6350, 1195] of gantry
      - frame TeachingPoints_08-08-01 at (8733.67, 11607.34, 288.56) mm, rotated rx 180 ry 0 rz 0 deg
        - target Point_08-08-01 (Cartesian target) at (0, 0, 0) mm; joints [8800, 6350, 1195] of gantry
      - frame TeachingPoints_09-08-01 at (9433.67, 11607.34, 288.56) mm, rotated rx 180 ry 0 rz 0 deg
        - target Point_09-08-01 (Cartesian target) at (0, 0, 0) mm; joints [9500, 6350, 1195] of gantry
      - frame TeachingPoints_10-08-01 at (10133.67, 11607.34, 288.56) mm, rotated rx 180 ry 0 rz 0 deg
        - target Point_10-08-01 (Cartesian target) at (0, 0, 0) mm; joints [10200, 6350, 1195] of gantry
      - frame TeachingPoints_11-08-01 at (10833.67, 11607.34, 288.56) mm, rotated rx 180 ry 0 rz 0 deg
        - target Point_11-08-01 (Cartesian target) at (0, 0, 0) mm; joints [10900, 6350, 1195] of gantry
      - frame TeachingPoints_12-08-01 at (11533.67, 11607.34, 288.56) mm, rotated rx 180 ry 0 rz 0 deg
        - target Point_12-08-01 (Cartesian target) at (0, 0, 0) mm; joints [11600, 6350, 1195] of gantry
      - frame TeachingPoints_13-08-01 at (12233.67, 11607.34, 288.56) mm, rotated rx 180 ry 0 rz 0 deg
        - target Point_13-08-01 (Cartesian target) at (0, 0, 0) mm; joints [12300, 6350, 1195] of gantry
      - frame TeachingPoints_14-08-01 at (12933.67, 11607.34, 288.56) mm, rotated rx 180 ry 0 rz 0 deg
        - target Point_14-08-01 (Cartesian target) at (0, 0, 0) mm; joints [13000, 6350, 1195] of gantry
      - frame TeachingPoints_15-08-01 at (13633.67, 11607.34, 288.56) mm, rotated rx 180 ry 0 rz 0 deg
        - target Point_15-08-01 (Cartesian target) at (0, 0, 0) mm; joints [13700, 6350, 1195] of gantry
      - frame TeachingPoints_16-08-01 at (14333.67, 11607.34, 288.56) mm, rotated rx 180 ry 0 rz 0 deg
        - target Point_16-08-01 (Cartesian target) at (0, 0, 0) mm; joints [14400, 6350, 1195] of gantry
      - frame TeachingPoints_17-08-01 at (15033.67, 11607.34, 288.56) mm, rotated rx 180 ry 0 rz 0 deg
        - target Point_17-08-01 (Cartesian target) at (0, 0, 0) mm; joints [15100, 6350, 1195] of gantry
      - frame TeachingPoints_18-08-01 at (15733.67, 11607.34, 288.56) mm, rotated rx 180 ry 0 rz 0 deg
        - target Point_18-08-01 (Cartesian target) at (0, 0, 0) mm; joints [15800, 6350, 1195] of gantry
      - frame TeachingPoints_19-08-01 at (16433.67, 11607.34, 288.56) mm, rotated rx 180 ry 0 rz 0 deg
        - target Point_19-08-01 (Cartesian target) at (0, 0, 0) mm; joints [16500, 6350, 1195] of gantry
      - frame TeachingPoints_20-08-01 at (17133.67, 11607.34, 288.56) mm, rotated rx 180 ry 0 rz 0 deg
        - target Point_20-08-01 (Cartesian target) at (0, 0, 0) mm; joints [17200, 6350, 1195] of gantry
      - frame TeachingPoints_01-09-01 at (3833.67, 10907.34, 288.56) mm, rotated rx 180 ry 0 rz 0 deg
        - target Point_01-09-01 (Cartesian target) at (0, 0, 0) mm; joints [3900, 7050, 1195] of gantry
      - frame TeachingPoints_02-09-01 at (4533.67, 10907.34, 288.56) mm, rotated rx 180 ry 0 rz 0 deg
        - target Point_02-09-01 (Cartesian target) at (0, 0, 0) mm; joints [4600, 7050, 1195] of gantry
      - frame TeachingPoints_03-09-01 at (5233.67, 10907.34, 288.56) mm, rotated rx 180 ry 0 rz 0 deg
        - target Point_03-09-01 (Cartesian target) at (0, 0, 0) mm; joints [5300, 7050, 1195] of gantry
      - frame TeachingPoints_04-09-01 at (5933.67, 10907.34, 288.56) mm, rotated rx 180 ry 0 rz 0 deg
        - target Point_04-09-01 (Cartesian target) at (0, 0, 0) mm; joints [6000, 7050, 1195] of gantry
      - frame TeachingPoints_05-09-01 at (6633.67, 10907.34, 288.56) mm, rotated rx 180 ry 0 rz 0 deg
        - target Point_05-09-01 (Cartesian target) at (0, 0, 0) mm; joints [6700, 7050, 1195] of gantry
      - frame TeachingPoints_06-09-01 at (7333.67, 10907.34, 288.56) mm, rotated rx 180 ry 0 rz 0 deg
        - target Point_06-09-01 (Cartesian target) at (0, 0, 0) mm; joints [7400, 7050, 1195] of gantry
      - frame TeachingPoints_07-09-01 at (8033.67, 10907.34, 288.56) mm, rotated rx 180 ry 0 rz 0 deg
        - target Point_07-09-01 (Cartesian target) at (0, 0, 0) mm; joints [8100, 7050, 1195] of gantry
      - frame TeachingPoints_08-09-01 at (8733.67, 10907.34, 288.56) mm, rotated rx 180 ry 0 rz 0 deg
        - target Point_08-09-01 (Cartesian target) at (0, 0, 0) mm; joints [8800, 7050, 1195] of gantry
      - frame TeachingPoints_09-09-01 at (9433.67, 10907.34, 288.56) mm, rotated rx 180 ry 0 rz 0 deg
        - target Point_09-09-01 (Cartesian target) at (0, 0, 0) mm; joints [9500, 7050, 1195] of gantry
      - frame TeachingPoints_10-09-01 at (10133.67, 10907.34, 288.56) mm, rotated rx 180 ry 0 rz 0 deg
        - target Point_10-09-01 (Cartesian target) at (0, 0, 0) mm; joints [10200, 7050, 1195] of gantry
      - frame TeachingPoints_11-09-01 at (10833.67, 10907.34, 288.56) mm, rotated rx 180 ry 0 rz 0 deg
        - target Point_11-09-01 (Cartesian target) at (0, 0, 0) mm; joints [10900, 7050, 1195] of gantry
      - frame TeachingPoints_12-09-01 at (11533.67, 10907.34, 288.56) mm, rotated rx 180 ry 0 rz 0 deg
        - target Point_12-09-01 (Cartesian target) at (0, 0, 0) mm; joints [11600, 7050, 1195] of gantry
      - frame TeachingPoints_13-09-01 at (12233.67, 10907.34, 288.56) mm, rotated rx 180 ry 0 rz 0 deg
        - target Point_13-09-01 (Cartesian target) at (0, 0, 0) mm; joints [12300, 7050, 1195] of gantry
      - frame TeachingPoints_14-09-01 at (12933.67, 10907.34, 288.56) mm, rotated rx 180 ry 0 rz 0 deg
        - target Point_14-09-01 (Cartesian target) at (0, 0, 0) mm; joints [13000, 7050, 1195] of gantry
      - frame TeachingPoints_15-09-01 at (13633.67, 10907.34, 288.56) mm, rotated rx 180 ry 0 rz 0 deg
        - target Point_15-09-01 (Cartesian target) at (0, 0, 0) mm; joints [13700, 7050, 1195] of gantry
      - frame TeachingPoints_16-09-01 at (14333.67, 10907.34, 288.56) mm, rotated rx 180 ry 0 rz 0 deg
        - target Point_16-09-01 (Cartesian target) at (0, 0, 0) mm; joints [14400, 7050, 1195] of gantry
      - frame TeachingPoints_17-09-01 at (15033.67, 10907.34, 288.56) mm, rotated rx 180 ry 0 rz 0 deg
        - target Point_17-09-01 (Cartesian target) at (0, 0, 0) mm; joints [15100, 7050, 1195] of gantry
      - frame TeachingPoints_18-09-01 at (15733.67, 10907.34, 288.56) mm, rotated rx 180 ry 0 rz 0 deg
        - target Point_18-09-01 (Cartesian target) at (0, 0, 0) mm; joints [15800, 7050, 1195] of gantry
      - frame TeachingPoints_19-09-01 at (16433.67, 10907.34, 288.56) mm, rotated rx 180 ry 0 rz 0 deg
        - target Point_19-09-01 (Cartesian target) at (0, 0, 0) mm; joints [16500, 7050, 1195] of gantry
      - frame TeachingPoints_20-09-01 at (17133.67, 10907.34, 288.56) mm, rotated rx 180 ry 0 rz 0 deg
        - target Point_20-09-01 (Cartesian target) at (0, 0, 0) mm; joints [17200, 7050, 1195] of gantry
      - frame TeachingPoints_01-10-01 at (3833.67, 10207.34, 288.56) mm, rotated rx 180 ry 0 rz 0 deg
        - target Point_01-10-01 (Cartesian target) at (0, 0, 0) mm; joints [3900, 7750, 1195] of gantry
      - frame TeachingPoints_02-10-01 at (4533.67, 10207.34, 288.56) mm, rotated rx 180 ry 0 rz 0 deg
        - target Point_02-10-01 (Cartesian target) at (0, 0, 0) mm; joints [4600, 7750, 1195] of gantry
      - frame TeachingPoints_03-10-01 at (5233.67, 10207.34, 288.56) mm, rotated rx 180 ry 0 rz 0 deg
        - target Point_03-10-01 (Cartesian target) at (0, 0, 0) mm; joints [5300, 7750, 1195] of gantry
      - frame TeachingPoints_04-10-01 at (5933.67, 10207.34, 288.56) mm, rotated rx 180 ry 0 rz 0 deg
        - target Point_04-10-01 (Cartesian target) at (0, 0, 0) mm; joints [6000, 7750, 1195] of gantry
      - frame TeachingPoints_05-10-01 at (6633.67, 10207.34, 288.56) mm, rotated rx 180 ry 0 rz 0 deg
        - target Point_05-10-01 (Cartesian target) at (0, 0, 0) mm; joints [6700, 7750, 1195] of gantry
      - frame TeachingPoints_06-10-01 at (7333.67, 10207.34, 288.56) mm, rotated rx 180 ry 0 rz 0 deg
        - target Point_06-10-01 (Cartesian target) at (0, 0, 0) mm; joints [7400, 7750, 1195] of gantry
      - frame TeachingPoints_07-10-01 at (8033.67, 10207.34, 288.56) mm, rotated rx 180 ry 0 rz 0 deg
        - target Point_07-10-01 (Cartesian target) at (0, 0, 0) mm; joints [8100, 7750, 1195] of gantry
      - frame TeachingPoints_08-10-01 at (8733.67, 10207.34, 288.56) mm, rotated rx 180 ry 0 rz 0 deg
        - target Point_08-10-01 (Cartesian target) at (0, 0, 0) mm; joints [8800, 7750, 1195] of gantry
      - frame TeachingPoints_09-10-01 at (9433.67, 10207.34, 288.56) mm, rotated rx 180 ry 0 rz 0 deg
        - target Point_09-10-01 (Cartesian target) at (0, 0, 0) mm; joints [9500, 7750, 1195] of gantry
      - frame TeachingPoints_10-10-01 at (10133.67, 10207.34, 288.56) mm, rotated rx 180 ry 0 rz 0 deg
        - target Point_10-10-01 (Cartesian target) at (0, 0, 0) mm; joints [10200, 7750, 1195] of gantry
      - frame TeachingPoints_11-10-01 at (10833.67, 10207.34, 288.56) mm, rotated rx 180 ry 0 rz 0 deg
        - target Point_11-10-01 (Cartesian target) at (0, 0, 0) mm; joints [10900, 7750, 1195] of gantry
      - frame TeachingPoints_12-10-01 at (11533.67, 10207.34, 288.56) mm, rotated rx 180 ry 0 rz 0 deg
        - target Point_12-10-01 (Cartesian target) at (0, 0, 0) mm; joints [11600, 7750, 1195] of gantry
      - frame TeachingPoints_13-10-01 at (12233.67, 10207.34, 288.56) mm, rotated rx 180 ry 0 rz 0 deg
        - target Point_13-10-01 (Cartesian target) at (0, 0, 0) mm; joints [12300, 7750, 1195] of gantry
      - frame TeachingPoints_14-10-01 at (12933.67, 10207.34, 288.56) mm, rotated rx 180 ry 0 rz 0 deg
        - target Point_14-10-01 (Cartesian target) at (0, 0, 0) mm; joints [13000, 7750, 1195] of gantry
      - frame TeachingPoints_15-10-01 at (13633.67, 10207.34, 288.56) mm, rotated rx 180 ry 0 rz 0 deg
        - target Point_15-10-01 (Cartesian target) at (0, 0, 0) mm; joints [13700, 7750, 1195] of gantry
      - frame TeachingPoints_16-10-01 at (14333.67, 10207.34, 288.56) mm, rotated rx 180 ry 0 rz 0 deg
        - target Point_16-10-01 (Cartesian target) at (0, 0, 0) mm; joints [14400, 7750, 1195] of gantry
      - frame TeachingPoints_17-10-01 at (15033.67, 10207.34, 288.56) mm, rotated rx 180 ry 0 rz 0 deg
        - target Point_17-10-01 (Cartesian target) at (0, 0, 0) mm; joints [15100, 7750, 1195] of gantry
      - frame TeachingPoints_18-10-01 at (15733.67, 10207.34, 288.56) mm, rotated rx 180 ry 0 rz 0 deg
        - target Point_18-10-01 (Cartesian target) at (0, 0, 0) mm; joints [15800, 7750, 1195] of gantry
      - frame TeachingPoints_19-10-01 at (16433.67, 10207.34, 288.56) mm, rotated rx 180 ry 0 rz 0 deg
        - target Point_19-10-01 (Cartesian target) at (0, 0, 0) mm; joints [16500, 7750, 1195] of gantry
      - frame TeachingPoints_20-10-01 at (17133.67, 10207.34, 288.56) mm, rotated rx 180 ry 0 rz 0 deg
        - target Point_20-10-01 (Cartesian target) at (0, 0, 0) mm; joints [17200, 7750, 1195] of gantry
      - frame TeachingPoints_01-11-01 at (3833.67, 9507.34, 288.56) mm, rotated rx 180 ry 0 rz 0 deg
        - target Point_01-11-01 (Cartesian target) at (0, 0, 0) mm; joints [3900, 8450, 1195] of gantry
      - frame TeachingPoints_02-11-01 at (4533.67, 9507.34, 288.56) mm, rotated rx 180 ry 0 rz 0 deg
        - target Point_02-11-01 (Cartesian target) at (0, 0, 0) mm; joints [4600, 8450, 1195] of gantry
      - frame TeachingPoints_03-11-01 at (5233.67, 9507.34, 288.56) mm, rotated rx 180 ry 0 rz 0 deg
        - target Point_03-11-01 (Cartesian target) at (0, 0, 0) mm; joints [5300, 8450, 1195] of gantry
      - frame TeachingPoints_04-11-01 at (5933.67, 9507.34, 288.56) mm, rotated rx 180 ry 0 rz 0 deg
        - target Point_04-11-01 (Cartesian target) at (0, 0, 0) mm; joints [6000, 8450, 1195] of gantry
      - frame TeachingPoints_05-11-01 at (6633.67, 9507.34, 288.56) mm, rotated rx 180 ry 0 rz 0 deg
        - target Point_05-11-01 (Cartesian target) at (0, 0, 0) mm; joints [6700, 8450, 1195] of gantry
      - frame TeachingPoints_06-11-01 at (7333.67, 9507.34, 288.56) mm, rotated rx 180 ry 0 rz 0 deg
        - target Point_06-11-01 (Cartesian target) at (0, 0, 0) mm; joints [7400, 8450, 1195] of gantry
      - frame TeachingPoints_07-11-01 at (8033.67, 9507.34, 288.56) mm, rotated rx 180 ry 0 rz 0 deg
        - target Point_07-11-01 (Cartesian target) at (0, 0, 0) mm; joints [8100, 8450, 1195] of gantry
      - frame TeachingPoints_08-11-01 at (8733.67, 9507.34, 288.56) mm, rotated rx 180 ry 0 rz 0 deg
        - target Point_08-11-01 (Cartesian target) at (0, 0, 0) mm; joints [8800, 8450, 1195] of gantry
      - frame TeachingPoints_09-11-01 at (9433.67, 9507.34, 288.56) mm, rotated rx 180 ry 0 rz 0 deg
        - target Point_09-11-01 (Cartesian target) at (0, 0, 0) mm; joints [9500, 8450, 1195] of gantry
      - frame TeachingPoints_10-11-01 at (10133.67, 9507.34, 288.56) mm, rotated rx 180 ry 0 rz 0 deg
        - target Point_10-11-01 (Cartesian target) at (0, 0, 0) mm; joints [10200, 8450, 1195] of gantry
      - frame TeachingPoints_11-11-01 at (10833.67, 9507.34, 288.56) mm, rotated rx 180 ry 0 rz 0 deg
        - target Point_11-11-01 (Cartesian target) at (0, 0, 0) mm; joints [10900, 8450, 1195] of gantry
      - frame TeachingPoints_12-11-01 at (11533.67, 9507.34, 288.56) mm, rotated rx 180 ry 0 rz 0 deg
        - target Point_12-11-01 (Cartesian target) at (0, 0, 0) mm; joints [11600, 8450, 1195] of gantry
      - frame TeachingPoints_13-11-01 at (12233.67, 9507.34, 288.56) mm, rotated rx 180 ry 0 rz 0 deg
        - target Point_13-11-01 (Cartesian target) at (0, 0, 0) mm; joints [12300, 8450, 1195] of gantry
      - frame TeachingPoints_14-11-01 at (12933.67, 9507.34, 288.56) mm, rotated rx 180 ry 0 rz 0 deg
        - target Point_14-11-01 (Cartesian target) at (0, 0, 0) mm; joints [13000, 8450, 1195] of gantry
      - frame TeachingPoints_15-11-01 at (13633.67, 9507.34, 288.56) mm, rotated rx 180 ry 0 rz 0 deg
        - target Point_15-11-01 (Cartesian target) at (0, 0, 0) mm; joints [13700, 8450, 1195] of gantry
      - frame TeachingPoints_16-11-01 at (14333.67, 9507.34, 288.56) mm, rotated rx 180 ry 0 rz 0 deg
        - target Point_16-11-01 (Cartesian target) at (0, 0, 0) mm; joints [14400, 8450, 1195] of gantry
      - frame TeachingPoints_17-11-01 at (15033.67, 9507.34, 288.56) mm, rotated rx 180 ry 0 rz 0 deg
        - target Point_17-11-01 (Cartesian target) at (0, 0, 0) mm; joints [15100, 8450, 1195] of gantry
      - frame TeachingPoints_18-11-01 at (15733.67, 9507.34, 288.56) mm, rotated rx 180 ry 0 rz 0 deg
        - target Point_18-11-01 (Cartesian target) at (0, 0, 0) mm; joints [15800, 8450, 1195] of gantry
      - frame TeachingPoints_19-11-01 at (16433.67, 9507.34, 288.56) mm, rotated rx 180 ry 0 rz 0 deg
        - target Point_19-11-01 (Cartesian target) at (0, 0, 0) mm; joints [16500, 8450, 1195] of gantry
      - frame TeachingPoints_20-11-01 at (17133.67, 9507.34, 288.56) mm, rotated rx 180 ry 0 rz 0 deg
        - target Point_20-11-01 (Cartesian target) at (0, 0, 0) mm; joints [17200, 8450, 1195] of gantry
      - frame TeachingPoints_01-12-01 at (3833.67, 8807.34, 288.56) mm, rotated rx 180 ry 0 rz 0 deg
        - target Point_01-12-01 (Cartesian target) at (0, 0, 0) mm; joints [3900, 9150, 1195] of gantry
      - frame TeachingPoints_02-12-01 at (4533.67, 8807.34, 288.56) mm, rotated rx 180 ry 0 rz 0 deg
        - target Point_02-12-01 (Cartesian target) at (0, 0, 0) mm; joints [4600, 9150, 1195] of gantry
      - frame TeachingPoints_03-12-01 at (5233.67, 8807.34, 288.56) mm, rotated rx 180 ry 0 rz 0 deg
        - target Point_03-12-01 (Cartesian target) at (0, 0, 0) mm; joints [5300, 9150, 1195] of gantry
      - frame TeachingPoints_04-12-01 at (5933.67, 8807.34, 288.56) mm, rotated rx 180 ry 0 rz 0 deg
        - target Point_04-12-01 (Cartesian target) at (0, 0, 0) mm; joints [6000, 9150, 1195] of gantry
      - frame TeachingPoints_05-12-01 at (6633.67, 8807.34, 288.56) mm, rotated rx 180 ry 0 rz 0 deg
        - target Point_05-12-01 (Cartesian target) at (0, 0, 0) mm; joints [6700, 9150, 1195] of gantry
      - frame TeachingPoints_06-12-01 at (7333.67, 8807.34, 288.56) mm, rotated rx 180 ry 0 rz 0 deg
        - target Point_06-12-01 (Cartesian target) at (0, 0, 0) mm; joints [7400, 9150, 1195] of gantry
      - frame TeachingPoints_07-12-01 at (8033.67, 8807.34, 288.56) mm, rotated rx 180 ry 0 rz 0 deg
        - target Point_07-12-01 (Cartesian target) at (0, 0, 0) mm; joints [8100, 9150, 1195] of gantry
      - frame TeachingPoints_08-12-01 at (8733.67, 8807.34, 288.56) mm, rotated rx 180 ry 0 rz 0 deg
        - target Point_08-12-01 (Cartesian target) at (0, 0, 0) mm; joints [8800, 9150, 1195] of gantry
      - frame TeachingPoints_09-12-01 at (9433.67, 8807.34, 288.56) mm, rotated rx 180 ry 0 rz 0 deg
        - target Point_09-12-01 (Cartesian target) at (0, 0, 0) mm; joints [9500, 9150, 1195] of gantry
      - frame TeachingPoints_10-12-01 at (10133.67, 8807.34, 288.56) mm, rotated rx 180 ry 0 rz 0 deg
        - target Point_10-12-01 (Cartesian target) at (0, 0, 0) mm; joints [10200, 9150, 1195] of gantry
      - frame TeachingPoints_11-12-01 at (10833.67, 8807.34, 288.56) mm, rotated rx 180 ry 0 rz 0 deg
        - target Point_11-12-01 (Cartesian target) at (0, 0, 0) mm; joints [10900, 9150, 1195] of gantry
      - frame TeachingPoints_12-12-01 at (11533.67, 8807.34, 288.56) mm, rotated rx 180 ry 0 rz 0 deg
        - target Point_12-12-01 (Cartesian target) at (0, 0, 0) mm; joints [11600, 9150, 1195] of gantry
      - frame TeachingPoints_13-12-01 at (12233.67, 8807.34, 288.56) mm, rotated rx 180 ry 0 rz 0 deg
        - target Point_13-12-01 (Cartesian target) at (0, 0, 0) mm; joints [12300, 9150, 1195] of gantry
      - frame TeachingPoints_14-12-01 at (12933.67, 8807.34, 288.56) mm, rotated rx 180 ry 0 rz 0 deg
        - target Point_14-12-01 (Cartesian target) at (0, 0, 0) mm; joints [13000, 9150, 1195] of gantry
      - frame TeachingPoints_15-12-01 at (13633.67, 8807.34, 288.56) mm, rotated rx 180 ry 0 rz 0 deg
        - target Point_15-12-01 (Cartesian target) at (0, 0, 0) mm; joints [13700, 9150, 1195] of gantry
      - frame TeachingPoints_16-12-01 at (14333.67, 8807.34, 288.56) mm, rotated rx 180 ry 0 rz 0 deg
        - target Point_16-12-01 (Cartesian target) at (0, 0, 0) mm; joints [14400, 9150, 1195] of gantry
      - frame TeachingPoints_17-12-01 at (15033.67, 8807.34, 288.56) mm, rotated rx 180 ry 0 rz 0 deg
        - target Point_17-12-01 (Cartesian target) at (0, 0, 0) mm; joints [15100, 9150, 1195] of gantry
      - frame TeachingPoints_18-12-01 at (15733.67, 8807.34, 288.56) mm, rotated rx 180 ry 0 rz 0 deg
        - target Point_18-12-01 (Cartesian target) at (0, 0, 0) mm; joints [15800, 9150, 1195] of gantry
      - frame TeachingPoints_19-12-01 at (16433.67, 8807.34, 288.56) mm, rotated rx 180 ry 0 rz 0 deg
        - target Point_19-12-01 (Cartesian target) at (0, 0, 0) mm; joints [16500, 9150, 1195] of gantry
      - frame TeachingPoints_20-12-01 at (17133.67, 8807.34, 288.56) mm, rotated rx 180 ry 0 rz 0 deg
        - target Point_20-12-01 (Cartesian target) at (0, 0, 0) mm; joints [17200, 9150, 1195] of gantry
      - frame TeachingPoints_01-13-01 at (3833.67, 8107.34, 288.56) mm, rotated rx 180 ry 0 rz 0 deg
        - target Point_01-13-01 (Cartesian target) at (0, 0, 0) mm; joints [3900, 9850, 1195] of gantry
      - frame TeachingPoints_02-13-01 at (4533.67, 8107.34, 288.56) mm, rotated rx 180 ry 0 rz 0 deg
        - target Point_02-13-01 (Cartesian target) at (0, 0, 0) mm; joints [4600, 9850, 1195] of gantry
      - frame TeachingPoints_03-13-01 at (5233.67, 8107.34, 288.56) mm, rotated rx 180 ry 0 rz 0 deg
        - target Point_03-13-01 (Cartesian target) at (0, 0, 0) mm; joints [5300, 9850, 1195] of gantry
      - frame TeachingPoints_04-13-01 at (5933.67, 8107.34, 288.56) mm, rotated rx 180 ry 0 rz 0 deg
        - target Point_04-13-01 (Cartesian target) at (0, 0, 0) mm; joints [6000, 9850, 1195] of gantry
      - frame TeachingPoints_05-13-01 at (6633.67, 8107.34, 288.56) mm, rotated rx 180 ry 0 rz 0 deg
        - target Point_05-13-01 (Cartesian target) at (0, 0, 0) mm; joints [6700, 9850, 1195] of gantry
      - frame TeachingPoints_06-13-01 at (7333.67, 8107.34, 288.56) mm, rotated rx 180 ry 0 rz 0 deg
        - target Point_06-13-01 (Cartesian target) at (0, 0, 0) mm; joints [7400, 9850, 1195] of gantry
      - frame TeachingPoints_07-13-01 at (8033.67, 8107.34, 288.56) mm, rotated rx 180 ry 0 rz 0 deg
        - target Point_07-13-01 (Cartesian target) at (0, 0, 0) mm; joints [8100, 9850, 1195] of gantry
      - frame TeachingPoints_08-13-01 at (8733.67, 8107.34, 288.56) mm, rotated rx 180 ry 0 rz 0 deg
        - target Point_08-13-01 (Cartesian target) at (0, 0, 0) mm; joints [8800, 9850, 1195] of gantry
      - frame TeachingPoints_09-13-01 at (9433.67, 8107.34, 288.56) mm, rotated rx 180 ry 0 rz 0 deg
        - target Point_09-13-01 (Cartesian target) at (0, 0, 0) mm; joints [9500, 9850, 1195] of gantry
      - frame TeachingPoints_10-13-01 at (10133.67, 8107.34, 288.56) mm, rotated rx 180 ry 0 rz 0 deg
        - target Point_10-13-01 (Cartesian target) at (0, 0, 0) mm; joints [10200, 9850, 1195] of gantry
      - frame TeachingPoints_11-13-01 at (10833.67, 8107.34, 288.56) mm, rotated rx 180 ry 0 rz 0 deg
        - target Point_11-13-01 (Cartesian target) at (0, 0, 0) mm; joints [10900, 9850, 1195] of gantry
      - frame TeachingPoints_12-13-01 at (11533.67, 8107.34, 288.56) mm, rotated rx 180 ry 0 rz 0 deg
        - target Point_12-13-01 (Cartesian target) at (0, 0, 0) mm; joints [11600, 9850, 1195] of gantry
      - frame TeachingPoints_13-13-01 at (12233.67, 8107.34, 288.56) mm, rotated rx 180 ry 0 rz 0 deg
        - target Point_13-13-01 (Cartesian target) at (0, 0, 0) mm; joints [12300, 9850, 1195] of gantry
      - frame TeachingPoints_14-13-01 at (12933.67, 8107.34, 288.56) mm, rotated rx 180 ry 0 rz 0 deg
        - target Point_14-13-01 (Cartesian target) at (0, 0, 0) mm; joints [13000, 9850, 1195] of gantry
      - frame TeachingPoints_15-13-01 at (13633.67, 8107.34, 288.56) mm, rotated rx 180 ry 0 rz 0 deg
        - target Point_15-13-01 (Cartesian target) at (0, 0, 0) mm; joints [13700, 9850, 1195] of gantry
      - frame TeachingPoints_16-13-01 at (14333.67, 8107.34, 288.56) mm, rotated rx 180 ry 0 rz 0 deg
        - target Point_16-13-01 (Cartesian target) at (0, 0, 0) mm; joints [14400, 9850, 1195] of gantry
      - frame TeachingPoints_17-13-01 at (15033.67, 8107.34, 288.56) mm, rotated rx 180 ry 0 rz 0 deg
        - target Point_17-13-01 (Cartesian target) at (0, 0, 0) mm; joints [15100, 9850, 1195] of gantry
      - frame TeachingPoints_18-13-01 at (15733.67, 8107.34, 288.56) mm, rotated rx 180 ry 0 rz 0 deg
        - target Point_18-13-01 (Cartesian target) at (0, 0, 0) mm; joints [15800, 9850, 1195] of gantry
      - frame TeachingPoints_19-13-01 at (16433.67, 8107.34, 288.56) mm, rotated rx 180 ry 0 rz 0 deg
        - target Point_19-13-01 (Cartesian target) at (0, 0, 0) mm; joints [16500, 9850, 1195] of gantry
      - frame TeachingPoints_20-13-01 at (17133.67, 8107.34, 288.56) mm, rotated rx 180 ry 0 rz 0 deg
        - target Point_20-13-01 (Cartesian target) at (0, 0, 0) mm; joints [17200, 9850, 1195] of gantry
      - frame TeachingPoints_01-14-01 at (3833.67, 7407.34, 288.56) mm, rotated rx 180 ry 0 rz 0 deg
        - target Point_01-14-01 (Cartesian target) at (0, 0, 0) mm; joints [3900, 10550, 1195] of gantry
      - frame TeachingPoints_02-14-01 at (4533.67, 7407.34, 288.56) mm, rotated rx 180 ry 0 rz 0 deg
        - target Point_02-14-01 (Cartesian target) at (0, 0, 0) mm; joints [4600, 10550, 1195] of gantry
      - frame TeachingPoints_03-14-01 at (5233.67, 7407.34, 288.56) mm, rotated rx 180 ry 0 rz 0 deg
        - target Point_03-14-01 (Cartesian target) at (0, 0, 0) mm; joints [5300, 10550, 1195] of gantry
      - frame TeachingPoints_04-14-01 at (5933.67, 7407.34, 288.56) mm, rotated rx 180 ry 0 rz 0 deg
        - target Point_04-14-01 (Cartesian target) at (0, 0, 0) mm; joints [6000, 10550, 1195] of gantry
      - frame TeachingPoints_05-14-01 at (6633.67, 7407.34, 288.56) mm, rotated rx 180 ry 0 rz 0 deg
        - target Point_05-14-01 (Cartesian target) at (0, 0, 0) mm; joints [6700, 10550, 1195] of gantry
      - frame TeachingPoints_06-14-01 at (7333.67, 7407.34, 288.56) mm, rotated rx 180 ry 0 rz 0 deg
        - target Point_06-14-01 (Cartesian target) at (0, 0, 0) mm; joints [7400, 10550, 1195] of gantry
      - frame TeachingPoints_07-14-01 at (8033.67, 7407.34, 288.56) mm, rotated rx 180 ry 0 rz 0 deg
        - target Point_07-14-01 (Cartesian target) at (0, 0, 0) mm; joints [8100, 10550, 1195] of gantry
      - frame TeachingPoints_08-14-01 at (8733.67, 7407.34, 288.56) mm, rotated rx 180 ry 0 rz 0 deg
        - target Point_08-14-01 (Cartesian target) at (0, 0, 0) mm; joints [8800, 10550, 1195] of gantry
      - frame TeachingPoints_09-14-01 at (9433.67, 7407.34, 288.56) mm, rotated rx 180 ry 0 rz 0 deg
        - target Point_09-14-01 (Cartesian target) at (0, 0, 0) mm; joints [9500, 10550, 1195] of gantry
      - frame TeachingPoints_10-14-01 at (10133.67, 7407.34, 288.56) mm, rotated rx 180 ry 0 rz 0 deg
        - target Point_10-14-01 (Cartesian target) at (0, 0, 0) mm; joints [10200, 10550, 1195] of gantry
      - frame TeachingPoints_11-14-01 at (10833.67, 7407.34, 288.56) mm, rotated rx 180 ry 0 rz 0 deg
        - target Point_11-14-01 (Cartesian target) at (0, 0, 0) mm; joints [10900, 10550, 1195] of gantry
      - frame TeachingPoints_12-14-01 at (11533.67, 7407.34, 288.56) mm, rotated rx 180 ry 0 rz 0 deg
        - target Point_12-14-01 (Cartesian target) at (0, 0, 0) mm; joints [11600, 10550, 1195] of gantry
      - frame TeachingPoints_13-14-01 at (12233.67, 7407.34, 288.56) mm, rotated rx 180 ry 0 rz 0 deg
        - target Point_13-14-01 (Cartesian target) at (0, 0, 0) mm; joints [12300, 10550, 1195] of gantry
      - frame TeachingPoints_14-14-01 at (12933.67, 7407.34, 288.56) mm, rotated rx 180 ry 0 rz 0 deg
        - target Point_14-14-01 (Cartesian target) at (0, 0, 0) mm; joints [13000, 10550, 1195] of gantry
      - frame TeachingPoints_15-14-01 at (13633.67, 7407.34, 288.56) mm, rotated rx 180 ry 0 rz 0 deg
        - target Point_15-14-01 (Cartesian target) at (0, 0, 0) mm; joints [13700, 10550, 1195] of gantry
      - frame TeachingPoints_16-14-01 at (14333.67, 7407.34, 288.56) mm, rotated rx 180 ry 0 rz 0 deg
        - target Point_16-14-01 (Cartesian target) at (0, 0, 0) mm; joints [14400, 10550, 1195] of gantry
      - frame TeachingPoints_17-14-01 at (15033.67, 7407.34, 288.56) mm, rotated rx 180 ry 0 rz 0 deg
        - target Point_17-14-01 (Cartesian target) at (0, 0, 0) mm; joints [15100, 10550, 1195] of gantry
      - frame TeachingPoints_18-14-01 at (15733.67, 7407.34, 288.56) mm, rotated rx 180 ry 0 rz 0 deg
        - target Point_18-14-01 (Cartesian target) at (0, 0, 0) mm; joints [15800, 10550, 1195] of gantry
      - frame TeachingPoints_19-14-01 at (16433.67, 7407.34, 288.56) mm, rotated rx 180 ry 0 rz 0 deg
        - target Point_19-14-01 (Cartesian target) at (0, 0, 0) mm; joints [16500, 10550, 1195] of gantry
      - frame TeachingPoints_20-14-01 at (17133.67, 7407.34, 288.56) mm, rotated rx 180 ry 0 rz 0 deg
        - target Point_20-14-01 (Cartesian target) at (0, 0, 0) mm; joints [17200, 10550, 1195] of gantry
      - frame TeachingPoints_01-15-01 at (3833.67, 6707.34, 288.56) mm, rotated rx 180 ry 0 rz 0 deg
        - target Point_01-15-01 (Cartesian target) at (0, 0, 0) mm; joints [3900, 11250, 1195] of gantry
      - frame TeachingPoints_02-15-01 at (4533.67, 6707.34, 288.56) mm, rotated rx 180 ry 0 rz 0 deg
        - target Point_02-15-01 (Cartesian target) at (0, 0, 0) mm; joints [4600, 11250, 1195] of gantry
      - frame TeachingPoints_03-15-01 at (5233.67, 6707.34, 288.56) mm, rotated rx 180 ry 0 rz 0 deg
        - target Point_03-15-01 (Cartesian target) at (0, 0, 0) mm; joints [5300, 11250, 1195] of gantry
      - frame TeachingPoints_04-15-01 at (5933.67, 6707.34, 288.56) mm, rotated rx 180 ry 0 rz 0 deg
        - target Point_04-15-01 (Cartesian target) at (0, 0, 0) mm; joints [6000, 11250, 1195] of gantry
      - frame TeachingPoints_05-15-01 at (6633.67, 6707.34, 288.56) mm, rotated rx 180 ry 0 rz 0 deg
        - target Point_05-15-01 (Cartesian target) at (0, 0, 0) mm; joints [6700, 11250, 1195] of gantry
      - frame TeachingPoints_06-15-01 at (7333.67, 6707.34, 288.56) mm, rotated rx 180 ry 0 rz 0 deg
        - target Point_06-15-01 (Cartesian target) at (0, 0, 0) mm; joints [7400, 11250, 1195] of gantry
      - frame TeachingPoints_07-15-01 at (8033.67, 6707.34, 288.56) mm, rotated rx 180 ry 0 rz 0 deg
        - target Point_07-15-01 (Cartesian target) at (0, 0, 0) mm; joints [8100, 11250, 1195] of gantry
      - frame TeachingPoints_08-15-01 at (8733.67, 6707.34, 288.56) mm, rotated rx 180 ry 0 rz 0 deg
        - target Point_08-15-01 (Cartesian target) at (0, 0, 0) mm; joints [8800, 11250, 1195] of gantry
      - frame TeachingPoints_09-15-01 at (9433.67, 6707.34, 288.56) mm, rotated rx 180 ry 0 rz 0 deg
        - target Point_09-15-01 (Cartesian target) at (0, 0, 0) mm; joints [9500, 11250, 1195] of gantry
      - frame TeachingPoints_10-15-01 at (10133.67, 6707.34, 288.56) mm, rotated rx 180 ry 0 rz 0 deg
        - target Point_10-15-01 (Cartesian target) at (0, 0, 0) mm; joints [10200, 11250, 1195] of gantry
      - frame TeachingPoints_11-15-01 at (10833.67, 6707.34, 288.56) mm, rotated rx 180 ry 0 rz 0 deg
        - target Point_11-15-01 (Cartesian target) at (0, 0, 0) mm; joints [10900, 11250, 1195] of gantry
      - frame TeachingPoints_12-15-01 at (11533.67, 6707.34, 288.56) mm, rotated rx 180 ry 0 rz 0 deg
        - target Point_12-15-01 (Cartesian target) at (0, 0, 0) mm; joints [11600, 11250, 1195] of gantry
      - frame TeachingPoints_13-15-01 at (12233.67, 6707.34, 288.56) mm, rotated rx 180 ry 0 rz 0 deg
        - target Point_13-15-01 (Cartesian target) at (0, 0, 0) mm; joints [12300, 11250, 1195] of gantry
      - frame TeachingPoints_14-15-01 at (12933.67, 6707.34, 288.56) mm, rotated rx 180 ry 0 rz 0 deg
        - target Point_14-15-01 (Cartesian target) at (0, 0, 0) mm; joints [13000, 11250, 1195] of gantry
      - frame TeachingPoints_15-15-01 at (13633.67, 6707.34, 288.56) mm, rotated rx 180 ry 0 rz 0 deg
        - target Point_15-15-01 (Cartesian target) at (0, 0, 0) mm; joints [13700, 11250, 1195] of gantry
      - frame TeachingPoints_16-15-01 at (14333.67, 6707.34, 288.56) mm, rotated rx 180 ry 0 rz 0 deg
        - target Point_16-15-01 (Cartesian target) at (0, 0, 0) mm; joints [14400, 11250, 1195] of gantry
      - frame TeachingPoints_17-15-01 at (15033.67, 6707.34, 288.56) mm, rotated rx 180 ry 0 rz 0 deg
        - target Point_17-15-01 (Cartesian target) at (0, 0, 0) mm; joints [15100, 11250, 1195] of gantry
      - frame TeachingPoints_18-15-01 at (15733.67, 6707.34, 288.56) mm, rotated rx 180 ry 0 rz 0 deg
        - target Point_18-15-01 (Cartesian target) at (0, 0, 0) mm; joints [15800, 11250, 1195] of gantry
      - frame TeachingPoints_19-15-01 at (16433.67, 6707.34, 288.56) mm, rotated rx 180 ry 0 rz 0 deg
        - target Point_19-15-01 (Cartesian target) at (0, 0, 0) mm; joints [16500, 11250, 1195] of gantry
      - frame TeachingPoints_20-15-01 at (17133.67, 6707.34, 288.56) mm, rotated rx 180 ry 0 rz 0 deg
        - target Point_20-15-01 (Cartesian target) at (0, 0, 0) mm; joints [17200, 11250, 1195] of gantry
      - frame TeachingPoints_01-16-01 at (3833.67, 6007.34, 288.56) mm, rotated rx 180 ry 0 rz 0 deg
        - target Point_01-16-01 (Cartesian target) at (0, 0, 0) mm; joints [3900, 11950, 1195] of gantry
      - frame TeachingPoints_02-16-01 at (4533.67, 6007.34, 288.56) mm, rotated rx 180 ry 0 rz 0 deg
        - target Point_02-16-01 (Cartesian target) at (0, 0, 0) mm; joints [4600, 11950, 1195] of gantry
      - frame TeachingPoints_03-16-01 at (5233.67, 6007.34, 288.56) mm, rotated rx 180 ry 0 rz 0 deg
        - target Point_03-16-01 (Cartesian target) at (0, 0, 0) mm; joints [5300, 11950, 1195] of gantry
      - frame TeachingPoints_04-16-01 at (5933.67, 6007.34, 288.56) mm, rotated rx 180 ry 0 rz 0 deg
        - target Point_04-16-01 (Cartesian target) at (0, 0, 0) mm; joints [6000, 11950, 1195] of gantry
      - frame TeachingPoints_05-16-01 at (6633.67, 6007.34, 288.56) mm, rotated rx 180 ry 0 rz 0 deg
        - target Point_05-16-01 (Cartesian target) at (0, 0, 0) mm; joints [6700, 11950, 1195] of gantry
      - frame TeachingPoints_06-16-01 at (7333.67, 6007.34, 288.56) mm, rotated rx 180 ry 0 rz 0 deg
        - target Point_06-16-01 (Cartesian target) at (0, 0, 0) mm; joints [7400, 11950, 1195] of gantry
      - frame TeachingPoints_07-16-01 at (8033.67, 6007.34, 288.56) mm, rotated rx 180 ry 0 rz 0 deg
        - target Point_07-16-01 (Cartesian target) at (0, 0, 0) mm; joints [8100, 11950, 1195] of gantry
      - frame TeachingPoints_08-16-01 at (8733.67, 6007.34, 288.56) mm, rotated rx 180 ry 0 rz 0 deg
        - target Point_08-16-01 (Cartesian target) at (0, 0, 0) mm; joints [8800, 11950, 1195] of gantry
      - frame TeachingPoints_09-16-01 at (9433.67, 6007.34, 288.56) mm, rotated rx 180 ry 0 rz 0 deg
        - target Point_09-16-01 (Cartesian target) at (0, 0, 0) mm; joints [9500, 11950, 1195] of gantry
      - frame TeachingPoints_10-16-01 at (10133.67, 6007.34, 288.56) mm, rotated rx 180 ry 0 rz 0 deg
        - target Point_10-16-01 (Cartesian target) at (0, 0, 0) mm; joints [10200, 11950, 1195] of gantry
      - frame TeachingPoints_11-16-01 at (10833.67, 6007.34, 288.56) mm, rotated rx 180 ry 0 rz 0 deg
        - target Point_11-16-01 (Cartesian target) at (0, 0, 0) mm; joints [10900, 11950, 1195] of gantry
      - frame TeachingPoints_12-16-01 at (11533.67, 6007.34, 288.56) mm, rotated rx 180 ry 0 rz 0 deg
        - target Point_12-16-01 (Cartesian target) at (0, 0, 0) mm; joints [11600, 11950, 1195] of gantry
      - frame TeachingPoints_13-16-01 at (12233.67, 6007.34, 288.56) mm, rotated rx 180 ry 0 rz 0 deg
        - target Point_13-16-01 (Cartesian target) at (0, 0, 0) mm; joints [12300, 11950, 1195] of gantry
      - frame TeachingPoints_14-16-01 at (12933.67, 6007.34, 288.56) mm, rotated rx 180 ry 0 rz 0 deg
        - target Point_14-16-01 (Cartesian target) at (0, 0, 0) mm; joints [13000, 11950, 1195] of gantry
      - frame TeachingPoints_15-16-01 at (13633.67, 6007.34, 288.56) mm, rotated rx 180 ry 0 rz 0 deg
        - target Point_15-16-01 (Cartesian target) at (0, 0, 0) mm; joints [13700, 11950, 1195] of gantry
      - frame TeachingPoints_16-16-01 at (14333.67, 6007.34, 288.56) mm, rotated rx 180 ry 0 rz 0 deg
        - target Point_16-16-01 (Cartesian target) at (0, 0, 0) mm; joints [14400, 11950, 1195] of gantry
      - frame TeachingPoints_17-16-01 at (15033.67, 6007.34, 288.56) mm, rotated rx 180 ry 0 rz 0 deg
        - target Point_17-16-01 (Cartesian target) at (0, 0, 0) mm; joints [15100, 11950, 1195] of gantry
      - frame TeachingPoints_18-16-01 at (15733.67, 6007.34, 288.56) mm, rotated rx 180 ry 0 rz 0 deg
        - target Point_18-16-01 (Cartesian target) at (0, 0, 0) mm; joints [15800, 11950, 1195] of gantry
      - frame TeachingPoints_19-16-01 at (16433.67, 6007.34, 288.56) mm, rotated rx 180 ry 0 rz 0 deg
        - target Point_19-16-01 (Cartesian target) at (0, 0, 0) mm; joints [16500, 11950, 1195] of gantry
      - frame TeachingPoints_20-16-01 at (17133.67, 6007.34, 288.56) mm, rotated rx 180 ry 0 rz 0 deg
        - target Point_20-16-01 (Cartesian target) at (0, 0, 0) mm; joints [17200, 11950, 1195] of gantry
      - frame TeachingPoints_01-17-01 at (3833.67, 5307.34, 288.56) mm, rotated rx 180 ry 0 rz 0 deg
        - target Point_01-17-01 (Cartesian target) at (0, 0, 0) mm; joints [3900, 12650, 1195] of gantry
      - frame TeachingPoints_02-17-01 at (4533.67, 5307.34, 288.56) mm, rotated rx 180 ry 0 rz 0 deg
        - target Point_02-17-01 (Cartesian target) at (0, 0, 0) mm; joints [4600, 12650, 1195] of gantry
      - frame TeachingPoints_03-17-01 at (5233.67, 5307.34, 288.56) mm, rotated rx 180 ry 0 rz 0 deg
        - target Point_03-17-01 (Cartesian target) at (0, 0, 0) mm; joints [5300, 12650, 1195] of gantry
      - frame TeachingPoints_04-17-01 at (5933.67, 5307.34, 288.56) mm, rotated rx 180 ry 0 rz 0 deg
        - target Point_04-17-01 (Cartesian target) at (0, 0, 0) mm; joints [6000, 12650, 1195] of gantry
      - frame TeachingPoints_05-17-01 at (6633.67, 5307.34, 288.56) mm, rotated rx 180 ry 0 rz 0 deg
        - target Point_05-17-01 (Cartesian target) at (0, 0, 0) mm; joints [6700, 12650, 1195] of gantry
      - frame TeachingPoints_06-17-01 at (7333.67, 5307.34, 288.56) mm, rotated rx 180 ry 0 rz 0 deg
        - target Point_06-17-01 (Cartesian target) at (0, 0, 0) mm; joints [7400, 12650, 1195] of gantry
      - frame TeachingPoints_07-17-01 at (8033.67, 5307.34, 288.56) mm, rotated rx 180 ry 0 rz 0 deg
        - target Point_07-17-01 (Cartesian target) at (0, 0, 0) mm; joints [8100, 12650, 1195] of gantry
      - frame TeachingPoints_08-17-01 at (8733.67, 5307.34, 288.56) mm, rotated rx 180 ry 0 rz 0 deg
        - target Point_08-17-01 (Cartesian target) at (0, 0, 0) mm; joints [8800, 12650, 1195] of gantry
      - frame TeachingPoints_09-17-01 at (9433.67, 5307.34, 288.56) mm, rotated rx 180 ry 0 rz 0 deg
        - target Point_09-17-01 (Cartesian target) at (0, 0, 0) mm; joints [9500, 12650, 1195] of gantry
      - frame TeachingPoints_10-17-01 at (10133.67, 5307.34, 288.56) mm, rotated rx 180 ry 0 rz 0 deg
        - target Point_10-17-01 (Cartesian target) at (0, 0, 0) mm; joints [10200, 12650, 1195] of gantry
      - frame TeachingPoints_11-17-01 at (10833.67, 5307.34, 288.56) mm, rotated rx 180 ry 0 rz 0 deg
        - target Point_11-17-01 (Cartesian target) at (0, 0, 0) mm; joints [10900, 12650, 1195] of gantry
      - frame TeachingPoints_12-17-01 at (11533.67, 5307.34, 288.56) mm, rotated rx 180 ry 0 rz 0 deg
        - target Point_12-17-01 (Cartesian target) at (0, 0, 0) mm; joints [11600, 12650, 1195] of gantry
      - frame TeachingPoints_13-17-01 at (12233.67, 5307.34, 288.56) mm, rotated rx 180 ry 0 rz 0 deg
        - target Point_13-17-01 (Cartesian target) at (0, 0, 0) mm; joints [12300, 12650, 1195] of gantry
      - frame TeachingPoints_14-17-01 at (12933.67, 5307.34, 288.56) mm, rotated rx 180 ry 0 rz 0 deg
        - target Point_14-17-01 (Cartesian target) at (0, 0, 0) mm; joints [13000, 12650, 1195] of gantry
      - frame TeachingPoints_15-17-01 at (13633.67, 5307.34, 288.56) mm, rotated rx 180 ry 0 rz 0 deg
        - target Point_15-17-01 (Cartesian target) at (0, 0, 0) mm; joints [13700, 12650, 1195] of gantry
      - frame TeachingPoints_16-17-01 at (14333.67, 5307.34, 288.56) mm, rotated rx 180 ry 0 rz 0 deg
        - target Point_16-17-01 (Cartesian target) at (0, 0, 0) mm; joints [14400, 12650, 1195] of gantry
      - frame TeachingPoints_17-17-01 at (15033.67, 5307.34, 288.56) mm, rotated rx 180 ry 0 rz 0 deg
        - target Point_17-17-01 (Cartesian target) at (0, 0, 0) mm; joints [15100, 12650, 1195] of gantry
      - frame TeachingPoints_18-17-01 at (15733.67, 5307.34, 288.56) mm, rotated rx 180 ry 0 rz 0 deg
        - target Point_18-17-01 (Cartesian target) at (0, 0, 0) mm; joints [15800, 12650, 1195] of gantry
      - frame TeachingPoints_19-17-01 at (16433.67, 5307.34, 288.56) mm, rotated rx 180 ry 0 rz 0 deg
        - target Point_19-17-01 (Cartesian target) at (0, 0, 0) mm; joints [16500, 12650, 1195] of gantry
      - frame TeachingPoints_20-17-01 at (17133.67, 5307.34, 288.56) mm, rotated rx 180 ry 0 rz 0 deg
        - target Point_20-17-01 (Cartesian target) at (0, 0, 0) mm; joints [17200, 12650, 1195] of gantry
      - frame TeachingPoints_01-18-01 at (3833.67, 4607.34, 288.56) mm, rotated rx 180 ry 0 rz 0 deg
        - target Point_01-18-01 (Cartesian target) at (0, 0, 0) mm; joints [3900, 13350, 1195] of gantry
      - frame TeachingPoints_02-18-01 at (4533.67, 4607.34, 288.56) mm, rotated rx 180 ry 0 rz 0 deg
        - target Point_02-18-01 (Cartesian target) at (0, 0, 0) mm; joints [4600, 13350, 1195] of gantry
      - frame TeachingPoints_03-18-01 at (5233.67, 4607.34, 288.56) mm, rotated rx 180 ry 0 rz 0 deg
        - target Point_03-18-01 (Cartesian target) at (0, 0, 0) mm; joints [5300, 13350, 1195] of gantry
      - frame TeachingPoints_04-18-01 at (5933.67, 4607.34, 288.56) mm, rotated rx 180 ry 0 rz 0 deg
        - target Point_04-18-01 (Cartesian target) at (0, 0, 0) mm; joints [6000, 13350, 1195] of gantry
      - frame TeachingPoints_05-18-01 at (6633.67, 4607.34, 288.56) mm, rotated rx 180 ry 0 rz 0 deg
        - target Point_05-18-01 (Cartesian target) at (0, 0, 0) mm; joints [6700, 13350, 1195] of gantry
      - frame TeachingPoints_06-18-01 at (7333.67, 4607.34, 288.56) mm, rotated rx 180 ry 0 rz 0 deg
        - target Point_06-18-01 (Cartesian target) at (0, 0, 0) mm; joints [7400, 13350, 1195] of gantry
      - frame TeachingPoints_07-18-01 at (8033.67, 4607.34, 288.56) mm, rotated rx 180 ry 0 rz 0 deg
        - target Point_07-18-01 (Cartesian target) at (0, 0, 0) mm; joints [8100, 13350, 1195] of gantry
      - frame TeachingPoints_08-18-01 at (8733.67, 4607.34, 288.56) mm, rotated rx 180 ry 0 rz 0 deg
        - target Point_08-18-01 (Cartesian target) at (0, 0, 0) mm; joints [8800, 13350, 1195] of gantry
      - frame TeachingPoints_09-18-01 at (9433.67, 4607.34, 288.56) mm, rotated rx 180 ry 0 rz 0 deg
        - target Point_09-18-01 (Cartesian target) at (0, 0, 0) mm; joints [9500, 13350, 1195] of gantry
      - frame TeachingPoints_10-18-01 at (10133.67, 4607.34, 288.56) mm, rotated rx 180 ry 0 rz 0 deg
        - target Point_10-18-01 (Cartesian target) at (0, 0, 0) mm; joints [10200, 13350, 1195] of gantry
      - frame TeachingPoints_11-18-01 at (10833.67, 4607.34, 288.56) mm, rotated rx 180 ry 0 rz 0 deg
        - target Point_11-18-01 (Cartesian target) at (0, 0, 0) mm; joints [10900, 13350, 1195] of gantry
      - frame TeachingPoints_12-18-01 at (11533.67, 4607.34, 288.56) mm, rotated rx 180 ry 0 rz 0 deg
        - target Point_12-18-01 (Cartesian target) at (0, 0, 0) mm; joints [11600, 13350, 1195] of gantry
      - frame TeachingPoints_13-18-01 at (12233.67, 4607.34, 288.56) mm, rotated rx 180 ry 0 rz 0 deg
        - target Point_13-18-01 (Cartesian target) at (0, 0, 0) mm; joints [12300, 13350, 1195] of gantry
      - frame TeachingPoints_14-18-01 at (12933.67, 4607.34, 288.56) mm, rotated rx 180 ry 0 rz 0 deg
        - target Point_14-18-01 (Cartesian target) at (0, 0, 0) mm; joints [13000, 13350, 1195] of gantry
      - frame TeachingPoints_15-18-01 at (13633.67, 4607.34, 288.56) mm, rotated rx 180 ry 0 rz 0 deg
        - target Point_15-18-01 (Cartesian target) at (0, 0, 0) mm; joints [13700, 13350, 1195] of gantry
      - frame TeachingPoints_16-18-01 at (14333.67, 4607.34, 288.56) mm, rotated rx 180 ry 0 rz 0 deg
        - target Point_16-18-01 (Cartesian target) at (0, 0, 0) mm; joints [14400, 13350, 1195] of gantry
      - frame TeachingPoints_17-18-01 at (15033.67, 4607.34, 288.56) mm, rotated rx 180 ry 0 rz 0 deg
        - target Point_17-18-01 (Cartesian target) at (0, 0, 0) mm; joints [15100, 13350, 1195] of gantry
      - frame TeachingPoints_18-18-01 at (15733.67, 4607.34, 288.56) mm, rotated rx 180 ry 0 rz 0 deg
        - target Point_18-18-01 (Cartesian target) at (0, 0, 0) mm; joints [15800, 13350, 1195] of gantry
      - frame TeachingPoints_19-18-01 at (16433.67, 4607.34, 288.56) mm, rotated rx 180 ry 0 rz 0 deg
        - target Point_19-18-01 (Cartesian target) at (0, 0, 0) mm; joints [16500, 13350, 1195] of gantry
      - frame TeachingPoints_20-18-01 at (17133.67, 4607.34, 288.56) mm, rotated rx 180 ry 0 rz 0 deg
        - target Point_20-18-01 (Cartesian target) at (0, 0, 0) mm; joints [17200, 13350, 1195] of gantry
      - frame TeachingPoints_01-19-01 at (3833.67, 3907.34, 288.56) mm, rotated rx 180 ry 0 rz 0 deg
        - target Point_01-19-01 (Cartesian target) at (0, 0, 0) mm; joints [3900, 14050, 1195] of gantry
      - frame TeachingPoints_02-19-01 at (4533.67, 3907.34, 288.56) mm, rotated rx 180 ry 0 rz 0 deg
        - target Point_02-19-01 (Cartesian target) at (0, 0, 0) mm; joints [4600, 14050, 1195] of gantry
      - frame TeachingPoints_03-19-01 at (5233.67, 3907.34, 288.56) mm, rotated rx 180 ry 0 rz 0 deg
        - target Point_03-19-01 (Cartesian target) at (0, 0, 0) mm; joints [5300, 14050, 1195] of gantry
      - frame TeachingPoints_04-19-01 at (5933.67, 3907.34, 288.56) mm, rotated rx 180 ry 0 rz 0 deg
        - target Point_04-19-01 (Cartesian target) at (0, 0, 0) mm; joints [6000, 14050, 1195] of gantry
      - frame TeachingPoints_05-19-01 at (6633.67, 3907.34, 288.56) mm, rotated rx 180 ry 0 rz 0 deg
        - target Point_05-19-01 (Cartesian target) at (0, 0, 0) mm; joints [6700, 14050, 1195] of gantry
      - frame TeachingPoints_06-19-01 at (7333.67, 3907.34, 288.56) mm, rotated rx 180 ry 0 rz 0 deg
        - target Point_06-19-01 (Cartesian target) at (0, 0, 0) mm; joints [7400, 14050, 1195] of gantry
      - frame TeachingPoints_07-19-01 at (8033.67, 3907.34, 288.56) mm, rotated rx 180 ry 0 rz 0 deg
        - target Point_07-19-01 (Cartesian target) at (0, 0, 0) mm; joints [8100, 14050, 1195] of gantry
      - frame TeachingPoints_08-19-01 at (8733.67, 3907.34, 288.56) mm, rotated rx 180 ry 0 rz 0 deg
        - target Point_08-19-01 (Cartesian target) at (0, 0, 0) mm; joints [8800, 14050, 1195] of gantry
      - frame TeachingPoints_09-19-01 at (9433.67, 3907.34, 288.56) mm, rotated rx 180 ry 0 rz 0 deg
        - target Point_09-19-01 (Cartesian target) at (0, 0, 0) mm; joints [9500, 14050, 1195] of gantry
      - frame TeachingPoints_10-19-01 at (10133.67, 3907.34, 288.56) mm, rotated rx 180 ry 0 rz 0 deg
        - target Point_10-19-01 (Cartesian target) at (0, 0, 0) mm; joints [10200, 14050, 1195] of gantry
      - frame TeachingPoints_11-19-01 at (10833.67, 3907.34, 288.56) mm, rotated rx 180 ry 0 rz 0 deg
        - target Point_11-19-01 (Cartesian target) at (0, 0, 0) mm; joints [10900, 14050, 1195] of gantry
      - frame TeachingPoints_12-19-01 at (11533.67, 3907.34, 288.56) mm, rotated rx 180 ry 0 rz 0 deg
        - target Point_12-19-01 (Cartesian target) at (0, 0, 0) mm; joints [11600, 14050, 1195] of gantry
      - frame TeachingPoints_13-19-01 at (12233.67, 3907.34, 288.56) mm, rotated rx 180 ry 0 rz 0 deg
        - target Point_13-19-01 (Cartesian target) at (0, 0, 0) mm; joints [12300, 14050, 1195] of gantry
      - frame TeachingPoints_14-19-01 at (12933.67, 3907.34, 288.56) mm, rotated rx 180 ry 0 rz 0 deg
        - target Point_14-19-01 (Cartesian target) at (0, 0, 0) mm; joints [13000, 14050, 1195] of gantry
      - frame TeachingPoints_15-19-01 at (13633.67, 3907.34, 288.56) mm, rotated rx 180 ry 0 rz 0 deg
        - target Point_15-19-01 (Cartesian target) at (0, 0, 0) mm; joints [13700, 14050, 1195] of gantry
      - frame TeachingPoints_16-19-01 at (14333.67, 3907.34, 288.56) mm, rotated rx 180 ry 0 rz 0 deg
        - target Point_16-19-01 (Cartesian target) at (0, 0, 0) mm; joints [14400, 14050, 1195] of gantry
      - frame TeachingPoints_17-19-01 at (15033.67, 3907.34, 288.56) mm, rotated rx 180 ry 0 rz 0 deg
        - target Point_17-19-01 (Cartesian target) at (0, 0, 0) mm; joints [15100, 14050, 1195] of gantry
      - frame TeachingPoints_18-19-01 at (15733.67, 3907.34, 288.56) mm, rotated rx 180 ry 0 rz 0 deg
        - target Point_18-19-01 (Cartesian target) at (0, 0, 0) mm; joints [15800, 14050, 1195] of gantry
      - frame TeachingPoints_19-19-01 at (16433.67, 3907.34, 288.56) mm, rotated rx 180 ry 0 rz 0 deg
        - target Point_19-19-01 (Cartesian target) at (0, 0, 0) mm; joints [16500, 14050, 1195] of gantry
      - frame TeachingPoints_20-19-01 at (17133.67, 3907.34, 288.56) mm, rotated rx 180 ry 0 rz 0 deg
        - target Point_20-19-01 (Cartesian target) at (0, 0, 0) mm; joints [17200, 14050, 1195] of gantry
      - frame TeachingPoints_01-20-01 at (3833.67, 3207.34, 288.56) mm, rotated rx 180 ry 0 rz 0 deg
        - target Point_01-20-01 (Cartesian target) at (0, 0, 0) mm; joints [3900, 14750, 1195] of gantry
      - frame TeachingPoints_02-20-01 at (4533.67, 3207.34, 288.56) mm, rotated rx 180 ry 0 rz 0 deg
        - target Point_02-20-01 (Cartesian target) at (0, 0, 0) mm; joints [4600, 14750, 1195] of gantry
      - frame TeachingPoints_03-20-01 at (5233.67, 3207.34, 288.56) mm, rotated rx 180 ry 0 rz 0 deg
        - target Point_03-20-01 (Cartesian target) at (0, 0, 0) mm; joints [5300, 14750, 1195] of gantry
      - frame TeachingPoints_04-20-01 at (5933.67, 3207.34, 288.56) mm, rotated rx 180 ry 0 rz 0 deg
        - target Point_04-20-01 (Cartesian target) at (0, 0, 0) mm; joints [6000, 14750, 1195] of gantry
      - frame TeachingPoints_05-20-01 at (6633.67, 3207.34, 288.56) mm, rotated rx 180 ry 0 rz 0 deg
        - target Point_05-20-01 (Cartesian target) at (0, 0, 0) mm; joints [6700, 14750, 1195] of gantry
      - frame TeachingPoints_06-20-01 at (7333.67, 3207.34, 288.56) mm, rotated rx 180 ry 0 rz 0 deg
        - target Point_06-20-01 (Cartesian target) at (0, 0, 0) mm; joints [7400, 14750, 1195] of gantry
      - frame TeachingPoints_07-20-01 at (8033.67, 3207.34, 288.56) mm, rotated rx 180 ry 0 rz 0 deg
        - target Point_07-20-01 (Cartesian target) at (0, 0, 0) mm; joints [8100, 14750, 1195] of gantry
      - frame TeachingPoints_08-20-01 at (8733.67, 3207.34, 288.56) mm, rotated rx 180 ry 0 rz 0 deg
        - target Point_08-20-01 (Cartesian target) at (0, 0, 0) mm; joints [8800, 14750, 1195] of gantry
      - frame TeachingPoints_09-20-01 at (9433.67, 3207.34, 288.56) mm, rotated rx 180 ry 0 rz 0 deg
        - target Point_09-20-01 (Cartesian target) at (0, 0, 0) mm; joints [9500, 14750, 1195] of gantry
      - frame TeachingPoints_10-20-01 at (10133.67, 3207.34, 288.56) mm, rotated rx 180 ry 0 rz 0 deg
        - target Point_10-20-01 (Cartesian target) at (0, 0, 0) mm; joints [10200, 14750, 1195] of gantry
      - frame TeachingPoints_11-20-01 at (10833.67, 3207.34, 288.56) mm, rotated rx 180 ry 0 rz 0 deg
        - target Point_11-20-01 (Cartesian target) at (0, 0, 0) mm; joints [10900, 14750, 1195] of gantry
      - frame TeachingPoints_12-20-01 at (11533.67, 3207.34, 288.56) mm, rotated rx 180 ry 0 rz 0 deg
        - target Point_12-20-01 (Cartesian target) at (0, 0, 0) mm; joints [11600, 14750, 1195] of gantry
      - frame TeachingPoints_13-20-01 at (12233.67, 3207.34, 288.56) mm, rotated rx 180 ry 0 rz 0 deg
        - target Point_13-20-01 (Cartesian target) at (0, 0, 0) mm; joints [12300, 14750, 1195] of gantry
      - frame TeachingPoints_14-20-01 at (12933.67, 3207.34, 288.56) mm, rotated rx 180 ry 0 rz 0 deg
        - target Point_14-20-01 (Cartesian target) at (0, 0, 0) mm; joints [13000, 14750, 1195] of gantry
      - frame TeachingPoints_15-20-01 at (13633.67, 3207.34, 288.56) mm, rotated rx 180 ry 0 rz 0 deg
        - target Point_15-20-01 (Cartesian target) at (0, 0, 0) mm; joints [13700, 14750, 1195] of gantry
      - frame TeachingPoints_16-20-01 at (14333.67, 3207.34, 288.56) mm, rotated rx 180 ry 0 rz 0 deg
        - target Point_16-20-01 (Cartesian target) at (0, 0, 0) mm; joints [14400, 14750, 1195] of gantry
      - frame TeachingPoints_17-20-01 at (15033.67, 3207.34, 288.56) mm, rotated rx 180 ry 0 rz 0 deg
        - target Point_17-20-01 (Cartesian target) at (0, 0, 0) mm; joints [15100, 14750, 1195] of gantry
      - frame TeachingPoints_18-20-01 at (15733.67, 3207.34, 288.56) mm, rotated rx 180 ry 0 rz 0 deg
        - target Point_18-20-01 (Cartesian target) at (0, 0, 0) mm; joints [15800, 14750, 1195] of gantry
      - frame TeachingPoints_19-20-01 at (16433.67, 3207.34, 288.56) mm, rotated rx 180 ry 0 rz 0 deg
        - target Point_19-20-01 (Cartesian target) at (0, 0, 0) mm; joints [16500, 14750, 1195] of gantry
      - frame TeachingPoints_20-20-01 at (17133.67, 3207.34, 288.56) mm, rotated rx 180 ry 0 rz 0 deg
        - target Point_20-20-01 (Cartesian target) at (0, 0, 0) mm; joints [17200, 14750, 1195] of gantry
      - frame TeachingPoints_01-01-02 at (3833.67, 16507.34, 423.56) mm, rotated rx 180 ry 0 rz 0 deg
        - target Point_01-01-02 (Cartesian target) at (0, 0, 0) mm; joints [3900, 1450, 1060] of gantry
      - frame TeachingPoints_02-01-02 at (4533.67, 16507.34, 423.56) mm, rotated rx 180 ry 0 rz 0 deg
        - target Point_02-01-02 (Cartesian target) at (0, 0, 0) mm; joints [4600, 1450, 1060] of gantry
      - frame TeachingPoints_03-01-02 at (5233.67, 16507.34, 423.56) mm, rotated rx 180 ry 0 rz 0 deg
        - target Point_03-01-02 (Cartesian target) at (0, 0, 0) mm; joints [5300, 1450, 1060] of gantry
      - frame TeachingPoints_04-01-02 at (5933.67, 16507.34, 423.56) mm, rotated rx 180 ry 0 rz 0 deg
        - target Point_04-01-02 (Cartesian target) at (0, 0, 0) mm; joints [6000, 1450, 1060] of gantry
      - frame TeachingPoints_05-01-02 at (6633.67, 16507.34, 423.56) mm, rotated rx 180 ry 0 rz 0 deg
        - target Point_05-01-02 (Cartesian target) at (0, 0, 0) mm; joints [6700, 1450, 1060] of gantry
      - frame TeachingPoints_06-01-02 at (7333.67, 16507.34, 423.56) mm, rotated rx 180 ry 0 rz 0 deg
        - target Point_06-01-02 (Cartesian target) at (0, 0, 0) mm; joints [7400, 1450, 1060] of gantry
      - frame TeachingPoints_07-01-02 at (8033.67, 16507.34, 423.56) mm, rotated rx 180 ry 0 rz 0 deg
        - target Point_07-01-02 (Cartesian target) at (0, 0, 0) mm; joints [8100, 1450, 1060] of gantry
      - frame TeachingPoints_08-01-02 at (8733.67, 16507.34, 423.56) mm, rotated rx 180 ry 0 rz 0 deg
        - target Point_08-01-02 (Cartesian target) at (0, 0, 0) mm; joints [8800, 1450, 1060] of gantry
      - frame TeachingPoints_09-01-02 at (9433.67, 16507.34, 423.56) mm, rotated rx 180 ry 0 rz 0 deg
        - target Point_09-01-02 (Cartesian target) at (0, 0, 0) mm; joints [9500, 1450, 1060] of gantry
      - frame TeachingPoints_10-01-02 at (10133.67, 16507.34, 423.56) mm, rotated rx 180 ry 0 rz 0 deg
        - target Point_10-01-02 (Cartesian target) at (0, 0, 0) mm; joints [10200, 1450, 1060] of gantry
      - frame TeachingPoints_11-01-02 at (10833.67, 16507.34, 423.56) mm, rotated rx 180 ry 0 rz 0 deg
        - target Point_11-01-02 (Cartesian target) at (0, 0, 0) mm; joints [10900, 1450, 1060] of gantry
      - frame TeachingPoints_12-01-02 at (11533.67, 16507.34, 423.56) mm, rotated rx 180 ry 0 rz 0 deg
        - target Point_12-01-02 (Cartesian target) at (0, 0, 0) mm; joints [11600, 1450, 1060] of gantry
      - frame TeachingPoints_13-01-02 at (12233.67, 16507.34, 423.56) mm, rotated rx 180 ry 0 rz 0 deg
        - target Point_13-01-02 (Cartesian target) at (0, 0, 0) mm; joints [12300, 1450, 1060] of gantry
      - frame TeachingPoints_14-01-02 at (12933.67, 16507.34, 423.56) mm, rotated rx 180 ry 0 rz 0 deg
        - target Point_14-01-02 (Cartesian target) at (0, 0, 0) mm; joints [13000, 1450, 1060] of gantry
      - frame TeachingPoints_15-01-02 at (13633.67, 16507.34, 423.56) mm, rotated rx 180 ry 0 rz 0 deg
        - target Point_15-01-02 (Cartesian target) at (0, 0, 0) mm; joints [13700, 1450, 1060] of gantry
      - frame TeachingPoints_16-01-02 at (14333.67, 16507.34, 423.56) mm, rotated rx 180 ry 0 rz 0 deg
        - target Point_16-01-02 (Cartesian target) at (0, 0, 0) mm; joints [14400, 1450, 1060] of gantry
      - frame TeachingPoints_17-01-02 at (15033.67, 16507.34, 423.56) mm, rotated rx 180 ry 0 rz 0 deg
        - target Point_17-01-02 (Cartesian target) at (0, 0, 0) mm; joints [15100, 1450, 1060] of gantry
      - frame TeachingPoints_18-01-02 at (15733.67, 16507.34, 423.56) mm, rotated rx 180 ry 0 rz 0 deg
        - target Point_18-01-02 (Cartesian target) at (0, 0, 0) mm; joints [15800, 1450, 1060] of gantry
      - frame TeachingPoints_19-01-02 at (16433.67, 16507.34, 423.56) mm, rotated rx 180 ry 0 rz 0 deg
        - target Point_19-01-02 (Cartesian target) at (0, 0, 0) mm; joints [16500, 1450, 1060] of gantry
      - frame TeachingPoints_20-01-02 at (17133.67, 16507.34, 423.56) mm, rotated rx 180 ry 0 rz 0 deg
        - target Point_20-01-02 (Cartesian target) at (0, 0, 0) mm; joints [17200, 1450, 1060] of gantry
      - frame TeachingPoints_01-02-02 at (3833.67, 15807.34, 423.56) mm, rotated rx 180 ry 0 rz 0 deg
        - target Point_01-02-02 (Cartesian target) at (0, 0, 0) mm; joints [3900, 2150, 1060] of gantry
      - frame TeachingPoints_02-02-02 at (4533.67, 15807.34, 423.56) mm, rotated rx 180 ry 0 rz 0 deg
        - target Point_02-02-02 (Cartesian target) at (0, 0, 0) mm; joints [4600, 2150, 1060] of gantry
      - frame TeachingPoints_03-02-02 at (5233.67, 15807.34, 423.56) mm, rotated rx 180 ry 0 rz 0 deg
        - target Point_03-02-02 (Cartesian target) at (0, 0, 0) mm; joints [5300, 2150, 1060] of gantry
      - frame TeachingPoints_04-02-02 at (5933.67, 15807.34, 423.56) mm, rotated rx 180 ry 0 rz 0 deg
        - target Point_04-02-02 (Cartesian target) at (0, 0, 0) mm; joints [6000, 2150, 1060] of gantry
      - frame TeachingPoints_05-02-02 at (6633.67, 15807.34, 423.56) mm, rotated rx 180 ry 0 rz 0 deg
        - target Point_05-02-02 (Cartesian target) at (0, 0, 0) mm; joints [6700, 2150, 1060] of gantry
      - frame TeachingPoints_06-02-02 at (7333.67, 15807.34, 423.56) mm, rotated rx 180 ry 0 rz 0 deg
        - target Point_06-02-02 (Cartesian target) at (0, 0, 0) mm; joints [7400, 2150, 1060] of gantry
      - frame TeachingPoints_07-02-02 at (8033.67, 15807.34, 423.56) mm, rotated rx 180 ry 0 rz 0 deg
        - target Point_07-02-02 (Cartesian target) at (0, 0, 0) mm; joints [8100, 2150, 1060] of gantry
      - frame TeachingPoints_08-02-02 at (8733.67, 15807.34, 423.56) mm, rotated rx 180 ry 0 rz 0 deg
        - target Point_08-02-02 (Cartesian target) at (0, 0, 0) mm; joints [8800, 2150, 1060] of gantry
      - frame TeachingPoints_09-02-02 at (9433.67, 15807.34, 423.56) mm, rotated rx 180 ry 0 rz 0 deg
        - target Point_09-02-02 (Cartesian target) at (0, 0, 0) mm; joints [9500, 2150, 1060] of gantry
      - frame TeachingPoints_10-02-02 at (10133.67, 15807.34, 423.56) mm, rotated rx 180 ry 0 rz 0 deg
        - target Point_10-02-02 (Cartesian target) at (0, 0, 0) mm; joints [10200, 2150, 1060] of gantry
      - frame TeachingPoints_11-02-02 at (10833.67, 15807.34, 423.56) mm, rotated rx 180 ry 0 rz 0 deg
        - target Point_11-02-02 (Cartesian target) at (0, 0, 0) mm; joints [10900, 2150, 1060] of gantry
      - frame TeachingPoints_12-02-02 at (11533.67, 15807.34, 423.56) mm, rotated rx 180 ry 0 rz 0 deg
        - target Point_12-02-02 (Cartesian target) at (0, 0, 0) mm; joints [11600, 2150, 1060] of gantry
      - frame TeachingPoints_13-02-02 at (12233.67, 15807.34, 423.56) mm, rotated rx 180 ry 0 rz 0 deg
        - target Point_13-02-02 (Cartesian target) at (0, 0, 0) mm; joints [12300, 2150, 1060] of gantry
      - frame TeachingPoints_14-02-02 at (12933.67, 15807.34, 423.56) mm, rotated rx 180 ry 0 rz 0 deg
        - target Point_14-02-02 (Cartesian target) at (0, 0, 0) mm; joints [13000, 2150, 1060] of gantry
      - frame TeachingPoints_15-02-02 at (13633.67, 15807.34, 423.56) mm, rotated rx 180 ry 0 rz 0 deg
        - target Point_15-02-02 (Cartesian target) at (0, 0, 0) mm; joints [13700, 2150, 1060] of gantry
      - frame TeachingPoints_16-02-02 at (14333.67, 15807.34, 423.56) mm, rotated rx 180 ry 0 rz 0 deg
        - target Point_16-02-02 (Cartesian target) at (0, 0, 0) mm; joints [14400, 2150, 1060] of gantry
      - frame TeachingPoints_17-02-02 at (15033.67, 15807.34, 423.56) mm, rotated rx 180 ry 0 rz 0 deg
        - target Point_17-02-02 (Cartesian target) at (0, 0, 0) mm; joints [15100, 2150, 1060] of gantry
      - frame TeachingPoints_18-02-02 at (15733.67, 15807.34, 423.56) mm, rotated rx 180 ry 0 rz 0 deg
        - target Point_18-02-02 (Cartesian target) at (0, 0, 0) mm; joints [15800, 2150, 1060] of gantry
      - frame TeachingPoints_19-02-02 at (16433.67, 15807.34, 423.56) mm, rotated rx 180 ry 0 rz 0 deg
        - target Point_19-02-02 (Cartesian target) at (0, 0, 0) mm; joints [16500, 2150, 1060] of gantry
      - frame TeachingPoints_20-02-02 at (17133.67, 15807.34, 423.56) mm, rotated rx 180 ry 0 rz 0 deg
        - target Point_20-02-02 (Cartesian target) at (0, 0, 0) mm; joints [17200, 2150, 1060] of gantry
      - frame TeachingPoints_01-03-02 at (3833.67, 15107.34, 423.56) mm, rotated rx 180 ry 0 rz 0 deg
        - target Point_01-03-02 (Cartesian target) at (0, 0, 0) mm; joints [3900, 2850, 1060] of gantry
      - frame TeachingPoints_02-03-02 at (4533.67, 15107.34, 423.56) mm, rotated rx 180 ry 0 rz 0 deg
        - target Point_02-03-02 (Cartesian target) at (0, 0, 0) mm; joints [4600, 2850, 1060] of gantry
      - frame TeachingPoints_03-03-02 at (5233.67, 15107.34, 423.56) mm, rotated rx 180 ry 0 rz 0 deg
        - target Point_03-03-02 (Cartesian target) at (0, 0, 0) mm; joints [5300, 2850, 1060] of gantry
      - frame TeachingPoints_04-03-02 at (5933.67, 15107.34, 423.56) mm, rotated rx 180 ry 0 rz 0 deg
        - target Point_04-03-02 (Cartesian target) at (0, 0, 0) mm; joints [6000, 2850, 1060] of gantry
      - frame TeachingPoints_05-03-02 at (6633.67, 15107.34, 423.56) mm, rotated rx 180 ry 0 rz 0 deg
        - target Point_05-03-02 (Cartesian target) at (0, 0, 0) mm; joints [6700, 2850, 1060] of gantry
      - frame TeachingPoints_06-03-02 at (7333.67, 15107.34, 423.56) mm, rotated rx 180 ry 0 rz 0 deg
        - target Point_06-03-02 (Cartesian target) at (0, 0, 0) mm; joints [7400, 2850, 1060] of gantry
      - frame TeachingPoints_07-03-02 at (8033.67, 15107.34, 423.56) mm, rotated rx 180 ry 0 rz 0 deg
        - target Point_07-03-02 (Cartesian target) at (0, 0, 0) mm; joints [8100, 2850, 1060] of gantry
      - frame TeachingPoints_08-03-02 at (8733.67, 15107.34, 423.56) mm, rotated rx 180 ry 0 rz 0 deg
        - target Point_08-03-02 (Cartesian target) at (0, 0, 0) mm; joints [8800, 2850, 1060] of gantry
      - frame TeachingPoints_09-03-02 at (9433.67, 15107.34, 423.56) mm, rotated rx 180 ry 0 rz 0 deg
        - target Point_09-03-02 (Cartesian target) at (0, 0, 0) mm; joints [9500, 2850, 1060] of gantry
      - frame TeachingPoints_10-03-02 at (10133.67, 15107.34, 423.56) mm, rotated rx 180 ry 0 rz 0 deg
        - target Point_10-03-02 (Cartesian target) at (0, 0, 0) mm; joints [10200, 2850, 1060] of gantry
      - frame TeachingPoints_11-03-02 at (10833.67, 15107.34, 423.56) mm, rotated rx 180 ry 0 rz 0 deg
        - target Point_11-03-02 (Cartesian target) at (0, 0, 0) mm; joints [10900, 2850, 1060] of gantry
      - frame TeachingPoints_12-03-02 at (11533.67, 15107.34, 423.56) mm, rotated rx 180 ry 0 rz 0 deg
        - target Point_12-03-02 (Cartesian target) at (0, 0, 0) mm; joints [11600, 2850, 1060] of gantry
      - frame TeachingPoints_13-03-02 at (12233.67, 15107.34, 423.56) mm, rotated rx 180 ry 0 rz 0 deg
        - target Point_13-03-02 (Cartesian target) at (0, 0, 0) mm; joints [12300, 2850, 1060] of gantry
      - frame TeachingPoints_14-03-02 at (12933.67, 15107.34, 423.56) mm, rotated rx 180 ry 0 rz 0 deg
        - target Point_14-03-02 (Cartesian target) at (0, 0, 0) mm; joints [13000, 2850, 1060] of gantry
      - frame TeachingPoints_15-03-02 at (13633.67, 15107.34, 423.56) mm, rotated rx 180 ry 0 rz 0 deg
        - target Point_15-03-02 (Cartesian target) at (0, 0, 0) mm; joints [13700, 2850, 1060] of gantry
      - frame TeachingPoints_16-03-02 at (14333.67, 15107.34, 423.56) mm, rotated rx 180 ry 0 rz 0 deg
        - target Point_16-03-02 (Cartesian target) at (0, 0, 0) mm; joints [14400, 2850, 1060] of gantry
      - frame TeachingPoints_17-03-02 at (15033.67, 15107.34, 423.56) mm, rotated rx 180 ry 0 rz 0 deg
        - target Point_17-03-02 (Cartesian target) at (0, 0, 0) mm; joints [15100, 2850, 1060] of gantry
      - frame TeachingPoints_18-03-02 at (15733.67, 15107.34, 423.56) mm, rotated rx 180 ry 0 rz 0 deg
        - target Point_18-03-02 (Cartesian target) at (0, 0, 0) mm; joints [15800, 2850, 1060] of gantry
      - frame TeachingPoints_19-03-02 at (16433.67, 15107.34, 423.56) mm, rotated rx 180 ry 0 rz 0 deg
        - target Point_19-03-02 (Cartesian target) at (0, 0, 0) mm; joints [16500, 2850, 1060] of gantry
      - frame TeachingPoints_20-03-02 at (17133.67, 15107.34, 423.56) mm, rotated rx 180 ry 0 rz 0 deg
        - target Point_20-03-02 (Cartesian target) at (0, 0, 0) mm; joints [17200, 2850, 1060] of gantry
      - frame TeachingPoints_01-04-02 at (3833.67, 14407.34, 423.56) mm, rotated rx 180 ry 0 rz 0 deg
        - target Point_01-04-02 (Cartesian target) at (0, 0, 0) mm; joints [3900, 3550, 1060] of gantry
      - frame TeachingPoints_02-04-02 at (4533.67, 14407.34, 423.56) mm, rotated rx 180 ry 0 rz 0 deg
        - target Point_02-04-02 (Cartesian target) at (0, 0, 0) mm; joints [4600, 3550, 1060] of gantry
      - frame TeachingPoints_03-04-02 at (5233.67, 14407.34, 423.56) mm, rotated rx 180 ry 0 rz 0 deg
        - target Point_03-04-02 (Cartesian target) at (0, 0, 0) mm; joints [5300, 3550, 1060] of gantry
      - frame TeachingPoints_04-04-02 at (5933.67, 14407.34, 423.56) mm, rotated rx 180 ry 0 rz 0 deg
        - target Point_04-04-02 (Cartesian target) at (0, 0, 0) mm; joints [6000, 3550, 1060] of gantry
      - frame TeachingPoints_05-04-02 at (6633.67, 14407.34, 423.56) mm, rotated rx 180 ry 0 rz 0 deg
        - target Point_05-04-02 (Cartesian target) at (0, 0, 0) mm; joints [6700, 3550, 1060] of gantry
      - frame TeachingPoints_06-04-02 at (7333.67, 14407.34, 423.56) mm, rotated rx 180 ry 0 rz 0 deg
        - target Point_06-04-02 (Cartesian target) at (0, 0, 0) mm; joints [7400, 3550, 1060] of gantry
      - frame TeachingPoints_07-04-02 at (8033.67, 14407.34, 423.56) mm, rotated rx 180 ry 0 rz 0 deg
        - target Point_07-04-02 (Cartesian target) at (0, 0, 0) mm; joints [8100, 3550, 1060] of gantry
      - frame TeachingPoints_08-04-02 at (8733.67, 14407.34, 423.56) mm, rotated rx 180 ry 0 rz 0 deg
        - target Point_08-04-02 (Cartesian target) at (0, 0, 0) mm; joints [8800, 3550, 1060] of gantry
      - frame TeachingPoints_09-04-02 at (9433.67, 14407.34, 423.56) mm, rotated rx 180 ry 0 rz 0 deg
        - target Point_09-04-02 (Cartesian target) at (0, 0, 0) mm; joints [9500, 3550, 1060] of gantry
      - frame TeachingPoints_10-04-02 at (10133.67, 14407.34, 423.56) mm, rotated rx 180 ry 0 rz 0 deg
        - target Point_10-04-02 (Cartesian target) at (0, 0, 0) mm; joints [10200, 3550, 1060] of gantry
      - frame TeachingPoints_11-04-02 at (10833.67, 14407.34, 423.56) mm, rotated rx 180 ry 0 rz 0 deg
        - target Point_11-04-02 (Cartesian target) at (0, 0, 0) mm; joints [10900, 3550, 1060] of gantry
      - frame TeachingPoints_12-04-02 at (11533.67, 14407.34, 423.56) mm, rotated rx 180 ry 0 rz 0 deg
